REGION Network 16: AV Outlet
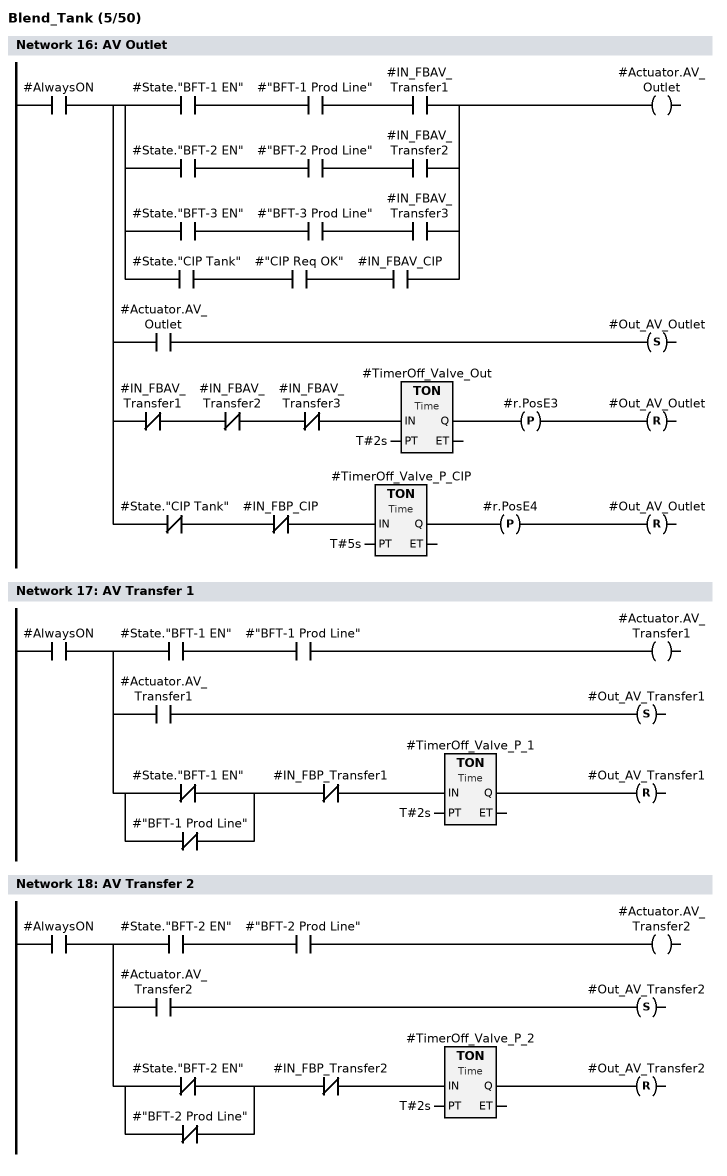
   RUNG wire#powerrail
      Contact( #AlwaysON )
      wire#w1
      Contact( #State."BFT-1 EN" )
      Contact( #"BFT-1 Prod Line" )
      Contact( #IN_FBAV_Transfer1 )
      wire#w2
      Coil( #Actuator.AV_Outlet )
   END_RUNG
   RUNG wire#w1
      Contact( #State."BFT-2 EN" )
      Contact( #"BFT-2 Prod Line" )
      Contact( #IN_FBAV_Transfer2 )
   END_RUNG wire#w2
   RUNG wire#w1
      Contact( #State."BFT-3 EN" )
      Contact( #"BFT-3 Prod Line" )
      Contact( #IN_FBAV_Transfer3 )
   END_RUNG wire#w2
   RUNG wire#w1
      Contact( #State."CIP Tank" )
      Contact( #"CIP Req OK" )
      Contact( #IN_FBAV_CIP )
   END_RUNG wire#w2
   RUNG wire#w1
      Contact( #Actuator.AV_Outlet )
      S_Coil( #Out_AV_Outlet )
   END_RUNG
   RUNG wire#w1
      I_Contact( #IN_FBAV_Transfer1 )
      I_Contact( #IN_FBAV_Transfer2 )
      I_Contact( #IN_FBAV_Transfer3 )
      { S7_Templates := "time_type := Time" } #TimerOff_Valve_Out.TON(pt := T#2s, et =>)
      P_Trig( #r.PosE3 )
      R_Coil( #Out_AV_Outlet )
   END_RUNG
   RUNG wire#w1
      I_Contact( #State."CIP Tank" )
      I_Contact( #IN_FBP_CIP )
      { S7_Templates := "time_type := Time" } #TimerOff_Valve_P_CIP.TON(pt := T#5s, et =>)
      P_Trig( #r.PosE4 )
      R_Coil( #Out_AV_Outlet )
   END_RUNG
   // the same network as SCL:
   #Actuator.AV_Outlet := #AlwaysON AND ((#State."BFT-1 EN" AND #"BFT-1 Prod Line" AND #IN_FBAV_Transfer1) OR (#State."BFT-2 EN" AND #"BFT-2 Prod Line" AND #IN_FBAV_Transfer2) OR (#State."BFT-3 EN" AND #"BFT-3 Prod Line" AND #IN_FBAV_Transfer3) OR (#State."CIP Tank" AND #"CIP Req OK" AND #IN_FBAV_CIP));
   IF #AlwaysON AND #Actuator.AV_Outlet THEN #Out_AV_Outlet := TRUE; END_IF;
   #TimerOff_Valve_Out(IN := #AlwaysON AND NOT #IN_FBAV_Transfer1 AND NOT #IN_FBAV_Transfer2 AND NOT #IN_FBAV_Transfer3,   // TON
                       PT := T#2s);
   #_w1 := #TimerOff_Valve_Out.Q AND NOT #r.PosE3;   // rising edge
   #r.PosE3 := #TimerOff_Valve_Out.Q;
   IF #_w1 THEN #Out_AV_Outlet := FALSE; END_IF;
   #TimerOff_Valve_P_CIP(IN := #AlwaysON AND NOT #State."CIP Tank" AND NOT #IN_FBP_CIP, PT := T#5s);   // TON
   #_w2 := #TimerOff_Valve_P_CIP.Q AND NOT #r.PosE4;   // rising edge
   #r.PosE4 := #TimerOff_Valve_P_CIP.Q;
   IF #_w2 THEN #Out_AV_Outlet := FALSE; END_IF;
END_REGION

REGION Network 17: AV Transfer 1
   RUNG wire#powerrail
      Contact( #AlwaysON )
      wire#w1
      Contact( #State."BFT-1 EN" )
      Contact( #"BFT-1 Prod Line" )
      Coil( #Actuator.AV_Transfer1 )
   END_RUNG
   RUNG wire#w1
      Contact( #Actuator.AV_Transfer1 )
      S_Coil( #Out_AV_Transfer1 )
   END_RUNG
   RUNG wire#w1
      I_Contact( #State."BFT-1 EN" )
      wire#w2
      I_Contact( #IN_FBP_Transfer1 )
      { S7_Templates := "time_type := Time" } #TimerOff_Valve_P_1.TON(pt := T#2s, et =>)
      R_Coil( #Out_AV_Transfer1 )
   END_RUNG
   RUNG wire#w1
      I_Contact( #"BFT-1 Prod Line" )
   END_RUNG wire#w2
   // the same network as SCL:
   #Actuator.AV_Transfer1 := #AlwaysON AND #State."BFT-1 EN" AND #"BFT-1 Prod Line";
   IF #AlwaysON AND #Actuator.AV_Transfer1 THEN #Out_AV_Transfer1 := TRUE; END_IF;
   #TimerOff_Valve_P_1(IN := #AlwaysON AND (NOT #State."BFT-1 EN" OR NOT #"BFT-1 Prod Line") AND NOT #IN_FBP_Transfer1,   // TON
                       PT := T#2s);
   IF #TimerOff_Valve_P_1.Q THEN #Out_AV_Transfer1 := FALSE; END_IF;
END_REGION

REGION Network 18: AV Transfer 2
   RUNG wire#powerrail
      Contact( #AlwaysON )
      wire#w1
      Contact( #State."BFT-2 EN" )
      Contact( #"BFT-2 Prod Line" )
      Coil( #Actuator.AV_Transfer2 )
   END_RUNG
   RUNG wire#w1
      Contact( #Actuator.AV_Transfer2 )
      S_Coil( #Out_AV_Transfer2 )
   END_RUNG
   RUNG wire#w1
      I_Contact( #State."BFT-2 EN" )
      wire#w2
      I_Contact( #IN_FBP_Transfer2 )
      { S7_Templates := "time_type := Time" } #TimerOff_Valve_P_2.TON(pt := T#2s, et =>)
      R_Coil( #Out_AV_Transfer2 )
   END_RUNG
   RUNG wire#w1
      I_Contact( #"BFT-2 Prod Line" )
   END_RUNG wire#w2
   // the same network as SCL:
   #Actuator.AV_Transfer2 := #AlwaysON AND #State."BFT-2 EN" AND #"BFT-2 Prod Line";
   IF #AlwaysON AND #Actuator.AV_Transfer2 THEN #Out_AV_Transfer2 := TRUE; END_IF;
   #TimerOff_Valve_P_2(IN := #AlwaysON AND (NOT #State."BFT-2 EN" OR NOT #"BFT-2 Prod Line") AND NOT #IN_FBP_Transfer2,   // TON
                       PT := T#2s);
   IF #TimerOff_Valve_P_2.Q THEN #Out_AV_Transfer2 := FALSE; END_IF;
END_REGION

REGION Network 19: AV Transfer 3
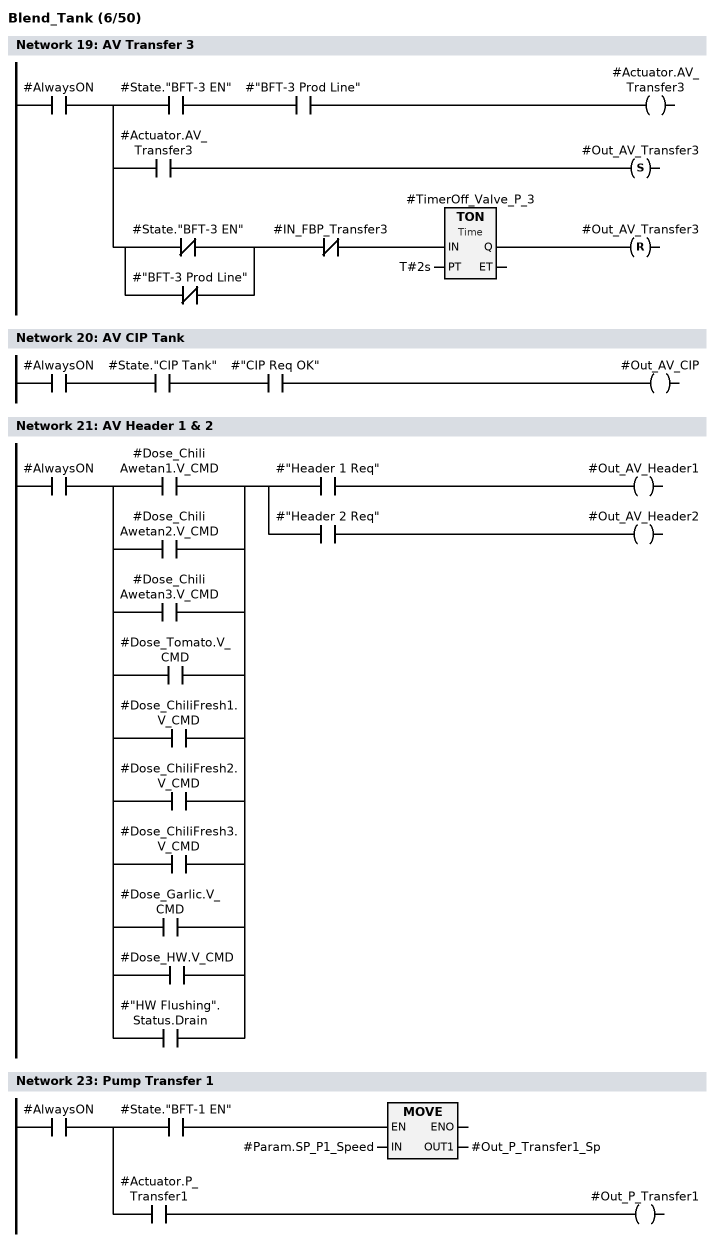
   RUNG wire#powerrail
      Contact( #AlwaysON )
      wire#w1
      Contact( #State."BFT-3 EN" )
      Contact( #"BFT-3 Prod Line" )
      Coil( #Actuator.AV_Transfer3 )
   END_RUNG
   RUNG wire#w1
      Contact( #Actuator.AV_Transfer3 )
      S_Coil( #Out_AV_Transfer3 )
   END_RUNG
   RUNG wire#w1
      I_Contact( #State."BFT-3 EN" )
      wire#w2
      I_Contact( #IN_FBP_Transfer3 )
      { S7_Templates := "time_type := Time" } #TimerOff_Valve_P_3.TON(pt := T#2s, et =>)
      R_Coil( #Out_AV_Transfer3 )
   END_RUNG
   RUNG wire#w1
      I_Contact( #"BFT-3 Prod Line" )
   END_RUNG wire#w2
   // the same network as SCL:
   #Actuator.AV_Transfer3 := #AlwaysON AND #State."BFT-3 EN" AND #"BFT-3 Prod Line";
   IF #AlwaysON AND #Actuator.AV_Transfer3 THEN #Out_AV_Transfer3 := TRUE; END_IF;
   #TimerOff_Valve_P_3(IN := #AlwaysON AND (NOT #State."BFT-3 EN" OR NOT #"BFT-3 Prod Line") AND NOT #IN_FBP_Transfer3,   // TON
                       PT := T#2s);
   IF #TimerOff_Valve_P_3.Q THEN #Out_AV_Transfer3 := FALSE; END_IF;
END_REGION

REGION Network 20: AV CIP Tank
   RUNG wire#powerrail
      Contact( #AlwaysON )
      Contact( #State."CIP Tank" )
      Contact( #"CIP Req OK" )
      Coil( #Out_AV_CIP )
   END_RUNG
   // the same network as SCL:
   #Out_AV_CIP := #AlwaysON AND #State."CIP Tank" AND #"CIP Req OK";
END_REGION

REGION Network 21: AV Header 1 & 2
   RUNG wire#powerrail
      Contact( #AlwaysON )
      wire#w1
      Contact( #Dose_ChiliAwetan1.V_CMD )
      wire#w2
      Contact( #"Header 1 Req" )
      Coil( #Out_AV_Header1 )
   END_RUNG
   RUNG wire#w1
      Contact( #Dose_ChiliAwetan2.V_CMD )
   END_RUNG wire#w2
   RUNG wire#w1
      Contact( #Dose_ChiliAwetan3.V_CMD )
   END_RUNG wire#w2
   RUNG wire#w1
      Contact( #Dose_Tomato.V_CMD )
   END_RUNG wire#w2
   RUNG wire#w1
      Contact( #Dose_ChiliFresh1.V_CMD )
   END_RUNG wire#w2
   RUNG wire#w1
      Contact( #Dose_ChiliFresh2.V_CMD )
   END_RUNG wire#w2
   RUNG wire#w1
      Contact( #Dose_ChiliFresh3.V_CMD )
   END_RUNG wire#w2
   RUNG wire#w1
      Contact( #Dose_Garlic.V_CMD )
   END_RUNG wire#w2
   RUNG wire#w1
      Contact( #Dose_HW.V_CMD )
   END_RUNG wire#w2
   RUNG wire#w1
      Contact( #"HW Flushing".Status.Drain )
   END_RUNG wire#w2
   RUNG wire#w2
      Contact( #"Header 2 Req" )
      Coil( #Out_AV_Header2 )
   END_RUNG
   // the same network as SCL:
   #_w1 := #AlwaysON AND (#Dose_ChiliAwetan1.V_CMD OR #Dose_ChiliAwetan2.V_CMD OR #Dose_ChiliAwetan3.V_CMD OR #Dose_Tomato.V_CMD OR #Dose_ChiliFresh1.V_CMD OR #Dose_ChiliFresh2.V_CMD OR #Dose_ChiliFresh3.V_CMD OR #Dose_Garlic.V_CMD OR #Dose_HW.V_CMD OR #"HW Flushing".Status.Drain);
   #Out_AV_Header1 := #_w1 AND #"Header 1 Req";
   #Out_AV_Header2 := #_w1 AND #"Header 2 Req";
END_REGION

REGION Network 23: Pump Transfer 1
   RUNG wire#powerrail
      Contact( #AlwaysON )
      wire#w1
      Contact( #State."BFT-1 EN" )
      Move(in := #Param.SP_P1_Speed, out1 => #Out_P_Transfer1_Sp)
   END_RUNG
   RUNG wire#w1
      Contact( #Actuator.P_Transfer1 )
      Coil( #Out_P_Transfer1 )
   END_RUNG
   // the same network as SCL:
   IF #AlwaysON AND #State."BFT-1 EN" THEN #Out_P_Transfer1_Sp := #Param.SP_P1_Speed; END_IF;
   #Out_P_Transfer1 := #AlwaysON AND #Actuator.P_Transfer1;
END_REGION

REGION Network 24: Pump Transfer 2
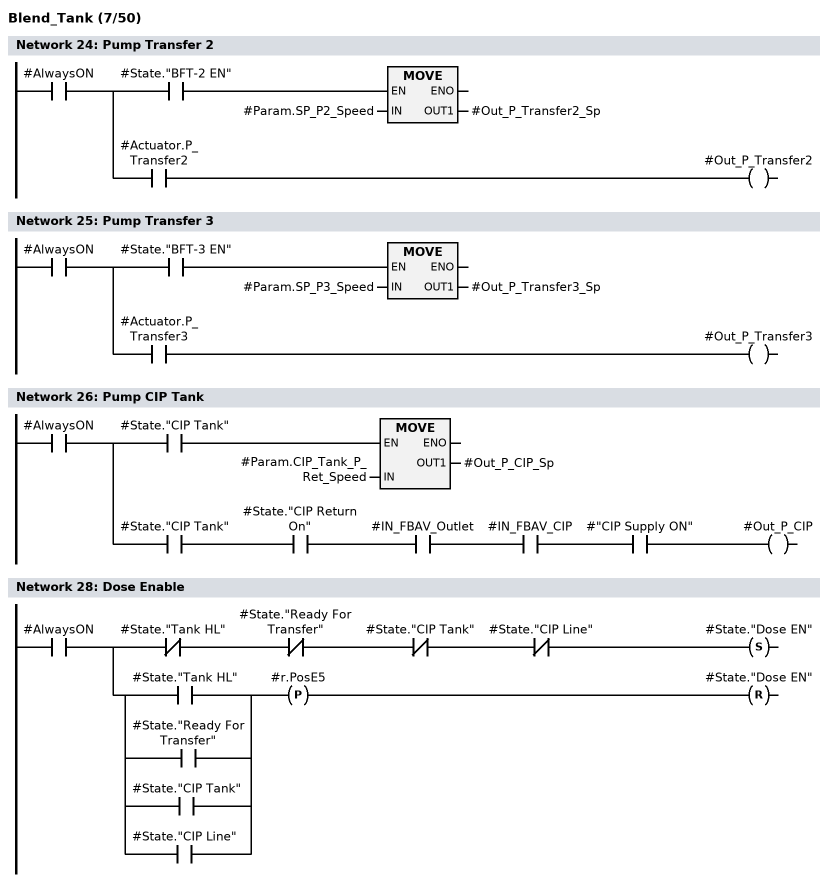
   RUNG wire#powerrail
      Contact( #AlwaysON )
      wire#w1
      Contact( #State."BFT-2 EN" )
      Move(in := #Param.SP_P2_Speed, out1 => #Out_P_Transfer2_Sp)
   END_RUNG
   RUNG wire#w1
      Contact( #Actuator.P_Transfer2 )
      Coil( #Out_P_Transfer2 )
   END_RUNG
   // the same network as SCL:
   IF #AlwaysON AND #State."BFT-2 EN" THEN #Out_P_Transfer2_Sp := #Param.SP_P2_Speed; END_IF;
   #Out_P_Transfer2 := #AlwaysON AND #Actuator.P_Transfer2;
END_REGION

REGION Network 25: Pump Transfer 3
   RUNG wire#powerrail
      Contact( #AlwaysON )
      wire#w1
      Contact( #State."BFT-3 EN" )
      Move(in := #Param.SP_P3_Speed, out1 => #Out_P_Transfer3_Sp)
   END_RUNG
   RUNG wire#w1
      Contact( #Actuator.P_Transfer3 )
      Coil( #Out_P_Transfer3 )
   END_RUNG
   // the same network as SCL:
   IF #AlwaysON AND #State."BFT-3 EN" THEN #Out_P_Transfer3_Sp := #Param.SP_P3_Speed; END_IF;
   #Out_P_Transfer3 := #AlwaysON AND #Actuator.P_Transfer3;
END_REGION

REGION Network 26: Pump CIP Tank
   RUNG wire#powerrail
      Contact( #AlwaysON )
      wire#w1
      Contact( #State."CIP Tank" )
      Move(in := #Param.CIP_Tank_P_Ret_Speed, out1 => #Out_P_CIP_Sp)
   END_RUNG
   RUNG wire#w1
      Contact( #State."CIP Tank" )
      Contact( #State."CIP Return On" )
      Contact( #IN_FBAV_Outlet )
      Contact( #IN_FBAV_CIP )
      Contact( #"CIP Supply ON" )
      Coil( #Out_P_CIP )
   END_RUNG
   // the same network as SCL:
   IF #AlwaysON AND #State."CIP Tank" THEN #Out_P_CIP_Sp := #Param.CIP_Tank_P_Ret_Speed; END_IF;
   #Out_P_CIP := #AlwaysON AND #State."CIP Tank" AND #State."CIP Return On" AND #IN_FBAV_Outlet AND #IN_FBAV_CIP AND #"CIP Supply ON";
END_REGION

REGION Network 28: Dose Enable
   RUNG wire#powerrail
      Contact( #AlwaysON )
      wire#w1
      I_Contact( #State."Tank HL" )
      I_Contact( #State."Ready For Transfer" )
      I_Contact( #State."CIP Tank" )
      I_Contact( #State."CIP Line" )
      S_Coil( #State."Dose EN" )
   END_RUNG
   RUNG wire#w1
      Contact( #State."Tank HL" )
      wire#w2
      P_Trig( #r.PosE5 )
      R_Coil( #State."Dose EN" )
   END_RUNG
   RUNG wire#w1
      Contact( #State."Ready For Transfer" )
   END_RUNG wire#w2
   RUNG wire#w1
      Contact( #State."CIP Tank" )
   END_RUNG wire#w2
   RUNG wire#w1
      Contact( #State."CIP Line" )
   END_RUNG wire#w2
   // the same network as SCL:
   IF #AlwaysON AND NOT #State."Tank HL" AND NOT #State."Ready For Transfer" AND NOT #State."CIP Tank" AND NOT #State."CIP Line" THEN
       #State."Dose EN" := TRUE;
   END_IF;
   #_w1 := #AlwaysON AND (#State."Tank HL" OR #State."Ready For Transfer" OR #State."CIP Tank" OR #State."CIP Line");
   #_w2 := #_w1 AND NOT #r.PosE5;   // rising edge
   #r.PosE5 := #_w1;
   IF #_w2 THEN #State."Dose EN" := FALSE; END_IF;
END_REGION

NETWORK
TITLE = Raw Material & Tank Dose State
// Raw Material Dose State
      O     #Dose_ChiliAwetan1.QDOSERun;
      O     #Dose_ChiliAwetan2.QDOSERun;
      O     #Dose_ChiliAwetan3.QDOSERun;
      O     #Dose_Tomato.QDOSERun;
      O     #Dose_ChiliFresh1.QDOSERun;
      O     #Dose_ChiliFresh2.QDOSERun;
      O     #Dose_ChiliFresh3.QDOSERun;
      O     #Dose_Garlic.QDOSERun;
      O     #Dose_HW.QDOSERun;
      =     #State."RM Dose";

// Dose Run State
      O     #State."RM Dose";
      O     #Dose_Vinegar.QDOSERun;
      O     #Dose_Sugar.QDOSERun;
      O     #Dose_Salt.QDOSERun;
      O     #Dose_ProWater.QDOSERun;
      O     #Dose_Homomixer.QDOSERun;
      =     #State."Dose On Prog";


REGION Network 31: Header 1 & 2 --- Vinegar --- Sugar --- Salt --- ProWater --- Homomixer Enable
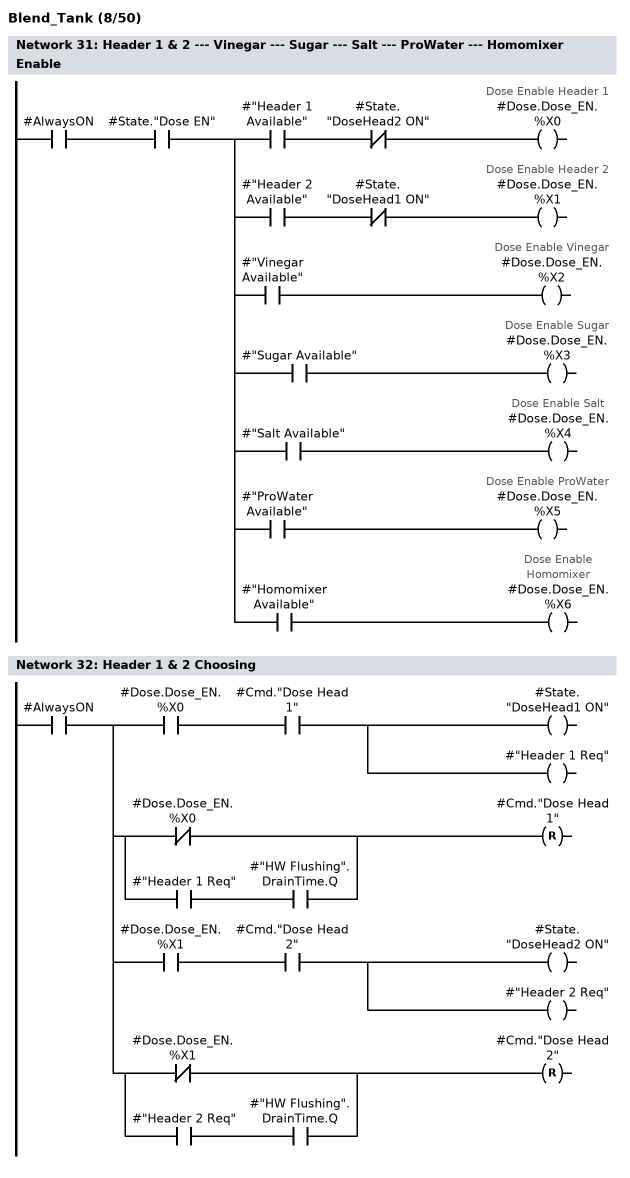
   RUNG wire#powerrail
      Contact( #AlwaysON )
      Contact( #State."Dose EN" )
      wire#w1
      Contact( #"Header 1 Available" )
      I_Contact( #State."DoseHead2 ON" )
      Coil( #Dose.Dose_EN.%X0 )   // Dose Enable Header 1
   END_RUNG
   RUNG wire#w1
      Contact( #"Header 2 Available" )
      I_Contact( #State."DoseHead1 ON" )
      Coil( #Dose.Dose_EN.%X1 )   // Dose Enable Header 2
   END_RUNG
   RUNG wire#w1
      Contact( #"Vinegar Available" )
      Coil( #Dose.Dose_EN.%X2 )   // Dose Enable Vinegar
   END_RUNG
   RUNG wire#w1
      Contact( #"Sugar Available" )
      Coil( #Dose.Dose_EN.%X3 )   // Dose Enable Sugar
   END_RUNG
   RUNG wire#w1
      Contact( #"Salt Available" )
      Coil( #Dose.Dose_EN.%X4 )   // Dose Enable Salt
   END_RUNG
   RUNG wire#w1
      Contact( #"ProWater Available" )
      Coil( #Dose.Dose_EN.%X5 )   // Dose Enable ProWater
   END_RUNG
   RUNG wire#w1
      Contact( #"Homomixer Available" )
      Coil( #Dose.Dose_EN.%X6 )   // Dose Enable Homomixer
   END_RUNG
   // the same network as SCL:
   #_w1 := #AlwaysON AND #State."Dose EN";
   #Dose.Dose_EN.%X0 := #_w1 AND #"Header 1 Available" AND NOT #State."DoseHead2 ON";   // Dose Enable Header 1
   #Dose.Dose_EN.%X1 := #_w1 AND #"Header 2 Available" AND NOT #State."DoseHead1 ON";   // Dose Enable Header 2
   #Dose.Dose_EN.%X2 := #_w1 AND #"Vinegar Available";   // Dose Enable Vinegar
   #Dose.Dose_EN.%X3 := #_w1 AND #"Sugar Available";   // Dose Enable Sugar
   #Dose.Dose_EN.%X4 := #_w1 AND #"Salt Available";   // Dose Enable Salt
   #Dose.Dose_EN.%X5 := #_w1 AND #"ProWater Available";   // Dose Enable ProWater
   #Dose.Dose_EN.%X6 := #_w1 AND #"Homomixer Available";   // Dose Enable Homomixer
END_REGION

REGION Network 32: Header 1 & 2 Choosing
   RUNG wire#powerrail
      Contact( #AlwaysON )
      wire#w1
      Contact( #Dose.Dose_EN.%X0 )
      Contact( #Cmd."Dose Head 1" )
      wire#w2
      Coil( #State."DoseHead1 ON" )
   END_RUNG
   RUNG wire#w2
      Coil( #"Header 1 Req" )
   END_RUNG
   RUNG wire#w1
      I_Contact( #Dose.Dose_EN.%X0 )
      wire#w3
      R_Coil( #Cmd."Dose Head 1" )
   END_RUNG
   RUNG wire#w1
      Contact( #"Header 1 Req" )
      Contact( #"HW Flushing".DrainTime.Q )
   END_RUNG wire#w3
   RUNG wire#w1
      Contact( #Dose.Dose_EN.%X1 )
      Contact( #Cmd."Dose Head 2" )
      wire#w4
      Coil( #State."DoseHead2 ON" )
   END_RUNG
   RUNG wire#w4
      Coil( #"Header 2 Req" )
   END_RUNG
   RUNG wire#w1
      I_Contact( #Dose.Dose_EN.%X1 )
      wire#w5
      R_Coil( #Cmd."Dose Head 2" )
   END_RUNG
   RUNG wire#w1
      Contact( #"Header 2 Req" )
      Contact( #"HW Flushing".DrainTime.Q )
   END_RUNG wire#w5
   // the same network as SCL:
   #State."DoseHead1 ON" := #AlwaysON AND #Dose.Dose_EN.%X0 AND #Cmd."Dose Head 1";
   #"Header 1 Req" := #State."DoseHead1 ON";
   IF #AlwaysON AND (NOT #Dose.Dose_EN.%X0 OR (#"Header 1 Req" AND #"HW Flushing".DrainTime.Q)) THEN
       #Cmd."Dose Head 1" := FALSE;
   END_IF;
   #State."DoseHead2 ON" := #AlwaysON AND #Dose.Dose_EN.%X1 AND #Cmd."Dose Head 2";
   #"Header 2 Req" := #State."DoseHead2 ON";
   IF #AlwaysON AND (NOT #Dose.Dose_EN.%X1 OR (#"Header 2 Req" AND #"HW Flushing".DrainTime.Q)) THEN
       #Cmd."Dose Head 2" := FALSE;
   END_IF;
END_REGION

NETWORK
TITLE = Header 1 & 2 Request
// Header 1 Request
//      O     #Dose.Dose_Header_Req.%X0// ChiliAwetan1 Header1 Req
//      O     #Dose.Dose_Header_Req.%X1// ChiliAwetan2 Header1 Req
//      O     #Dose.Dose_Header_Req.%X2// ChiliAwetan3 Header1 Req
//      O     #Dose.Dose_Header_Req.%X3// Tomato Header1 Req
//      O     #Dose.Dose_Header_Req.%X4// ChiliFresh1 Header1 Req
//      O     #Dose.Dose_Header_Req.%X5// ChiliFresh2 Header1 Req
//      O     #Dose.Dose_Header_Req.%X6// ChiliFresh3 Header1 Req
//      O     #Dose.Dose_Header_Req.%X7// Garlic Header1 Req
//      O     #Dose.Dose_Header_Req.%X8// HotWater Header1 Req
//     =     #"Header 1 Req"

// Header 2 Request
//      O     #Dose.Dose_Header_Req.%X16// ChiliAwetan1 Header2 Req
//      O     #Dose.Dose_Header_Req.%X17// ChiliAwetan2 Header2 Req
//      O     #Dose.Dose_Header_Req.%X18// ChiliAwetan3 Header2 Req
//      O     #Dose.Dose_Header_Req.%X19// Tomato Header2 Req
//      O     #Dose.Dose_Header_Req.%X20// ChiliFresh1 Header2 Req
//      O     #Dose.Dose_Header_Req.%X21// ChiliFresh2 Header2 Req
//      O     #Dose.Dose_Header_Req.%X22// ChiliFresh3 Header2 Req
//      O     #Dose.Dose_Header_Req.%X23// Garlic Header2 Req
//      O     #Dose.Dose_Header_Req.%X24// HotWater Header2 Req
//      =     #"Header 2 Req"


REGION Network 36: ChiliAwetan1 Setpoint
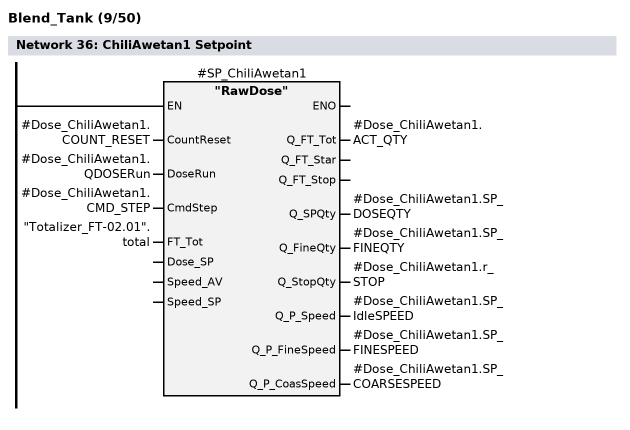
   RUNG wire#powerrail
      #SP_ChiliAwetan1(CountReset := #Dose_ChiliAwetan1.COUNT_RESET, DoseRun := #Dose_ChiliAwetan1.QDOSERun, CmdStep := #Dose_ChiliAwetan1.CMD_STEP, FT_Tot := "Totalizer_FT-02.01".total, Dose_SP :=, Speed_AV :=, Speed_SP :=, Q_FT_Tot => #Dose_ChiliAwetan1.ACT_QTY, Q_FT_Star =>, Q_FT_Stop =>, Q_SPQty => #Dose_ChiliAwetan1.SP_DOSEQTY, Q_FineQty => #Dose_ChiliAwetan1.SP_FINEQTY, Q_StopQty => #Dose_ChiliAwetan1.r_STOP, Q_P_Speed => #Dose_ChiliAwetan1.SP_IdleSPEED, Q_P_FineSpeed => #Dose_ChiliAwetan1.SP_FINESPEED, Q_P_CoasSpeed => #Dose_ChiliAwetan1.SP_COARSESPEED)
   END_RUNG
   // the same network as SCL:
   #SP_ChiliAwetan1(CountReset := #Dose_ChiliAwetan1.COUNT_RESET,   // "RawDose"
                    DoseRun := #Dose_ChiliAwetan1.QDOSERun,
                    CmdStep := #Dose_ChiliAwetan1.CMD_STEP,
                    FT_Tot := "Totalizer_FT-02.01".total,
                    Q_FT_Tot => #Dose_ChiliAwetan1.ACT_QTY,
                    Q_SPQty => #Dose_ChiliAwetan1.SP_DOSEQTY,
                    Q_FineQty => #Dose_ChiliAwetan1.SP_FINEQTY,
                    Q_StopQty => #Dose_ChiliAwetan1.r_STOP,
                    Q_P_Speed => #Dose_ChiliAwetan1.SP_IdleSPEED,
                    Q_P_FineSpeed => #Dose_ChiliAwetan1.SP_FINESPEED,
                    Q_P_CoasSpeed => #Dose_ChiliAwetan1.SP_COARSESPEED);
END_REGION

REGION Network 37: Command Dose ChiliAwetan1
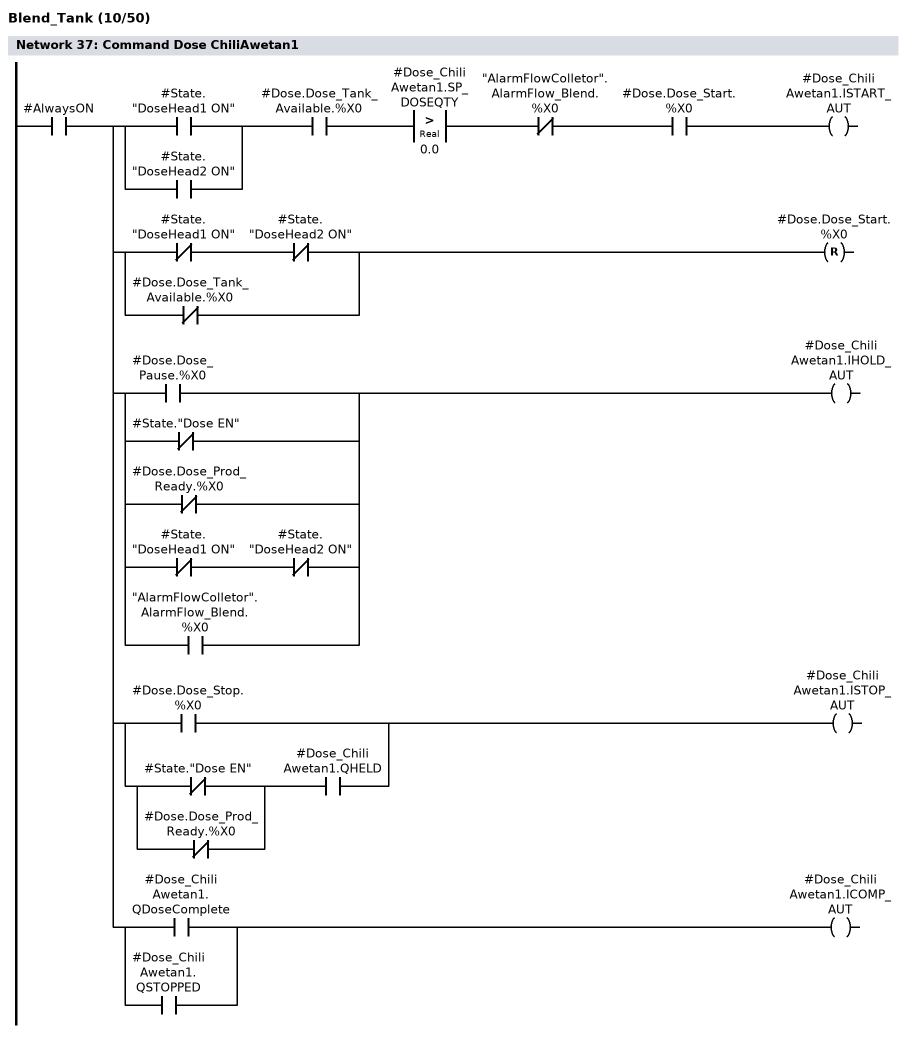
   RUNG wire#powerrail
      Contact( #AlwaysON )
      wire#w1
      Contact( #State."DoseHead1 ON" )
      wire#w2
      Contact( #Dose.Dose_Tank_Available.%X0 )
      { S7_Templates := "SrcType := Real" } GT_Contact(in1 := #Dose_ChiliAwetan1.SP_DOSEQTY, in2 := 0.0)
      I_Contact( "AlarmFlowColletor".AlarmFlow_Blend.%X0 )
      Contact( #Dose.Dose_Start.%X0 )
      Coil( #Dose_ChiliAwetan1.ISTART_AUT )
   END_RUNG
   RUNG wire#w1
      Contact( #State."DoseHead2 ON" )
   END_RUNG wire#w2
   RUNG wire#w1
      I_Contact( #State."DoseHead1 ON" )
      I_Contact( #State."DoseHead2 ON" )
      wire#w3
      R_Coil( #Dose.Dose_Start.%X0 )
   END_RUNG
   RUNG wire#w1
      I_Contact( #Dose.Dose_Tank_Available.%X0 )
   END_RUNG wire#w3
   RUNG wire#w1
      Contact( #Dose.Dose_Pause.%X0 )
      wire#w4
      Coil( #Dose_ChiliAwetan1.IHOLD_AUT )
   END_RUNG
   RUNG wire#w1
      I_Contact( #State."Dose EN" )
   END_RUNG wire#w4
   RUNG wire#w1
      I_Contact( #Dose.Dose_Prod_Ready.%X0 )
   END_RUNG wire#w4
   RUNG wire#w1
      I_Contact( #State."DoseHead1 ON" )
      I_Contact( #State."DoseHead2 ON" )
   END_RUNG wire#w4
   RUNG wire#w1
      Contact( "AlarmFlowColletor".AlarmFlow_Blend.%X0 )
   END_RUNG wire#w4
   RUNG wire#w1
      Contact( #Dose.Dose_Stop.%X0 )
      wire#w5
      Coil( #Dose_ChiliAwetan1.ISTOP_AUT )
   END_RUNG
   RUNG wire#w1
      I_Contact( #State."Dose EN" )
      wire#w6
      Contact( #Dose_ChiliAwetan1.QHELD )
   END_RUNG wire#w5
   RUNG wire#w1
      I_Contact( #Dose.Dose_Prod_Ready.%X0 )
   END_RUNG wire#w6
   RUNG wire#w1
      Contact( #Dose_ChiliAwetan1.QDoseComplete )
      wire#w7
      Coil( #Dose_ChiliAwetan1.ICOMP_AUT )
   END_RUNG
   RUNG wire#w1
      Contact( #Dose_ChiliAwetan1.QSTOPPED )
   END_RUNG wire#w7
   // the same network as SCL:
   #Dose_ChiliAwetan1.ISTART_AUT := #AlwaysON AND (#State."DoseHead1 ON" OR #State."DoseHead2 ON") AND #Dose.Dose_Tank_Available.%X0 AND (#Dose_ChiliAwetan1.SP_DOSEQTY > 0.0) AND NOT "AlarmFlowColletor".AlarmFlow_Blend.%X0 AND #Dose.Dose_Start.%X0;
   IF #AlwaysON AND ((NOT #State."DoseHead1 ON" AND NOT #State."DoseHead2 ON") OR NOT #Dose.Dose_Tank_Available.%X0) THEN
       #Dose.Dose_Start.%X0 := FALSE;
   END_IF;
   #Dose_ChiliAwetan1.IHOLD_AUT := #AlwaysON AND (#Dose.Dose_Pause.%X0 OR NOT #State."Dose EN" OR NOT #Dose.Dose_Prod_Ready.%X0 OR (NOT #State."DoseHead1 ON" AND NOT #State."DoseHead2 ON") OR "AlarmFlowColletor".AlarmFlow_Blend.%X0);
   #Dose_ChiliAwetan1.ISTOP_AUT := #AlwaysON AND (#Dose.Dose_Stop.%X0 OR ((NOT #State."Dose EN" OR NOT #Dose.Dose_Prod_Ready.%X0) AND #Dose_ChiliAwetan1.QHELD));
   #Dose_ChiliAwetan1.ICOMP_AUT := #AlwaysON AND (#Dose_ChiliAwetan1.QDoseComplete OR #Dose_ChiliAwetan1.QSTOPPED);
END_REGION

REGION Network 38: Dose ChiliAwetan1
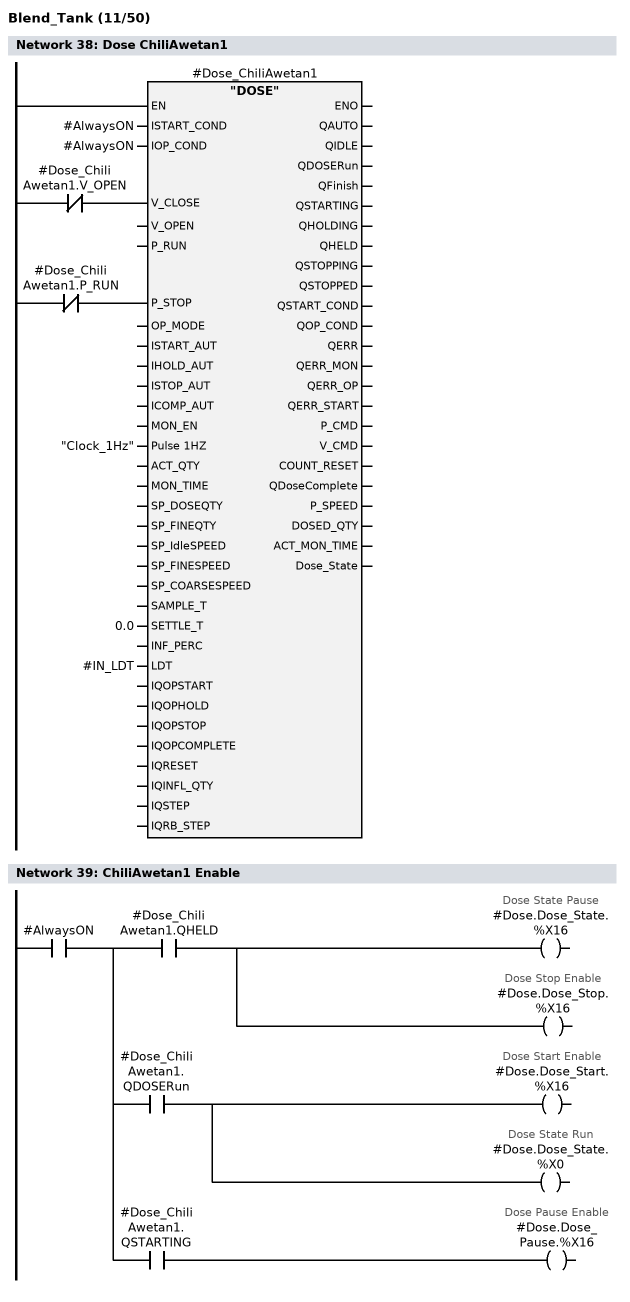
   RUNG wire#powerrail
      #Dose_ChiliAwetan1(V_CLOSE := wire#w1, P_STOP := wire#w2, ISTART_COND := #AlwaysON, IOP_COND := #AlwaysON, V_OPEN :=, P_RUN :=, OP_MODE :=, ISTART_AUT :=, IHOLD_AUT :=, ISTOP_AUT :=, ICOMP_AUT :=, MON_EN :=, "Pulse 1HZ" := "Clock_1Hz", ACT_QTY :=, MON_TIME :=, SP_DOSEQTY :=, SP_FINEQTY :=, SP_IdleSPEED :=, SP_FINESPEED :=, SP_COARSESPEED :=, SAMPLE_T :=, SETTLE_T := 0.0, INF_PERC :=, LDT := #IN_LDT, IQOPSTART :=, IQOPHOLD :=, IQOPSTOP :=, IQOPCOMPLETE :=, IQRESET :=, IQINFL_QTY :=, IQSTEP :=, IQRB_STEP :=, QAUTO =>, QIDLE =>, QDOSERun =>, QFinish =>, QSTARTING =>, QHOLDING =>, QHELD =>, QSTOPPING =>, QSTOPPED =>, QSTART_COND =>, QOP_COND =>, QERR =>, QERR_MON =>, QERR_OP =>, QERR_START =>, P_CMD =>, V_CMD =>, COUNT_RESET =>, QDoseComplete =>, P_SPEED =>, DOSED_QTY =>, ACT_MON_TIME =>, Dose_State =>)
   END_RUNG
   RUNG wire#powerrail
      I_Contact( #Dose_ChiliAwetan1.V_OPEN )
   END_RUNG wire#w1
   RUNG wire#powerrail
      I_Contact( #Dose_ChiliAwetan1.P_RUN )
   END_RUNG wire#w2
   // the same network as SCL:
   #Dose_ChiliAwetan1(ISTART_COND := #AlwaysON,   // "DOSE"
                      IOP_COND := #AlwaysON,
                      V_CLOSE := NOT #Dose_ChiliAwetan1.V_OPEN,
                      P_STOP := NOT #Dose_ChiliAwetan1.P_RUN,
                      "Pulse 1HZ" := "Clock_1Hz",
                      SETTLE_T := 0.0,
                      LDT := #IN_LDT);
END_REGION

REGION Network 39: ChiliAwetan1 Enable
   RUNG wire#powerrail
      Contact( #AlwaysON )
      wire#w1
      Contact( #Dose_ChiliAwetan1.QHELD )
      wire#w2
      Coil( #Dose.Dose_State.%X16 )   // Dose State Pause
   END_RUNG
   RUNG wire#w2
      Coil( #Dose.Dose_Stop.%X16 )   // Dose Stop Enable
   END_RUNG
   RUNG wire#w1
      Contact( #Dose_ChiliAwetan1.QDOSERun )
      wire#w3
      Coil( #Dose.Dose_Start.%X16 )   // Dose Start Enable
   END_RUNG
   RUNG wire#w3
      Coil( #Dose.Dose_State.%X0 )   // Dose State Run
   END_RUNG
   RUNG wire#w1
      Contact( #Dose_ChiliAwetan1.QSTARTING )
      Coil( #Dose.Dose_Pause.%X16 )   // Dose Pause Enable
   END_RUNG
   // the same network as SCL:
   #Dose.Dose_State.%X16 := #AlwaysON AND #Dose_ChiliAwetan1.QHELD;   // Dose State Pause
   #Dose.Dose_Stop.%X16 := #Dose.Dose_State.%X16;   // Dose Stop Enable
   #Dose.Dose_Start.%X16 := #AlwaysON AND #Dose_ChiliAwetan1.QDOSERun;   // Dose Start Enable
   #Dose.Dose_State.%X0 := #Dose.Dose_Start.%X16;   // Dose State Run
   #Dose.Dose_Pause.%X16 := #AlwaysON AND #Dose_ChiliAwetan1.QSTARTING;   // Dose Pause Enable
END_REGION

REGION Network 40: ChiliAwetan1 Header Req
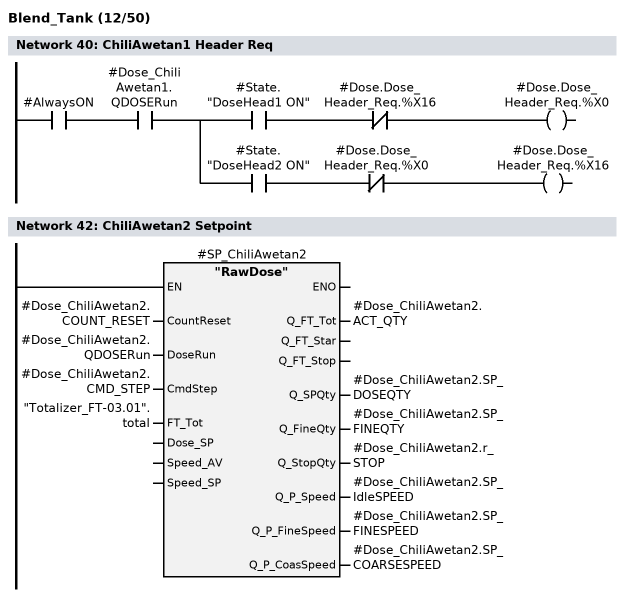
   RUNG wire#powerrail
      Contact( #AlwaysON )
      Contact( #Dose_ChiliAwetan1.QDOSERun )
      wire#w1
      Contact( #State."DoseHead1 ON" )
      I_Contact( #Dose.Dose_Header_Req.%X16 )
      Coil( #Dose.Dose_Header_Req.%X0 )
   END_RUNG
   RUNG wire#w1
      Contact( #State."DoseHead2 ON" )
      I_Contact( #Dose.Dose_Header_Req.%X0 )
      Coil( #Dose.Dose_Header_Req.%X16 )
   END_RUNG
   // the same network as SCL:
   #_w1 := #AlwaysON AND #Dose_ChiliAwetan1.QDOSERun;
   #Dose.Dose_Header_Req.%X0 := #_w1 AND #State."DoseHead1 ON" AND NOT #Dose.Dose_Header_Req.%X16;
   #Dose.Dose_Header_Req.%X16 := #_w1 AND #State."DoseHead2 ON" AND NOT #Dose.Dose_Header_Req.%X0;
END_REGION

REGION Network 42: ChiliAwetan2 Setpoint
   RUNG wire#powerrail
      #SP_ChiliAwetan2(CountReset := #Dose_ChiliAwetan2.COUNT_RESET, DoseRun := #Dose_ChiliAwetan2.QDOSERun, CmdStep := #Dose_ChiliAwetan2.CMD_STEP, FT_Tot := "Totalizer_FT-03.01".total, Dose_SP :=, Speed_AV :=, Speed_SP :=, Q_FT_Tot => #Dose_ChiliAwetan2.ACT_QTY, Q_FT_Star =>, Q_FT_Stop =>, Q_SPQty => #Dose_ChiliAwetan2.SP_DOSEQTY, Q_FineQty => #Dose_ChiliAwetan2.SP_FINEQTY, Q_StopQty => #Dose_ChiliAwetan2.r_STOP, Q_P_Speed => #Dose_ChiliAwetan2.SP_IdleSPEED, Q_P_FineSpeed => #Dose_ChiliAwetan2.SP_FINESPEED, Q_P_CoasSpeed => #Dose_ChiliAwetan2.SP_COARSESPEED)
   END_RUNG
   // the same network as SCL:
   #SP_ChiliAwetan2(CountReset := #Dose_ChiliAwetan2.COUNT_RESET,   // "RawDose"
                    DoseRun := #Dose_ChiliAwetan2.QDOSERun,
                    CmdStep := #Dose_ChiliAwetan2.CMD_STEP,
                    FT_Tot := "Totalizer_FT-03.01".total,
                    Q_FT_Tot => #Dose_ChiliAwetan2.ACT_QTY,
                    Q_SPQty => #Dose_ChiliAwetan2.SP_DOSEQTY,
                    Q_FineQty => #Dose_ChiliAwetan2.SP_FINEQTY,
                    Q_StopQty => #Dose_ChiliAwetan2.r_STOP,
                    Q_P_Speed => #Dose_ChiliAwetan2.SP_IdleSPEED,
                    Q_P_FineSpeed => #Dose_ChiliAwetan2.SP_FINESPEED,
                    Q_P_CoasSpeed => #Dose_ChiliAwetan2.SP_COARSESPEED);
END_REGION

REGION Network 43: Command Dose ChiliAwetan2
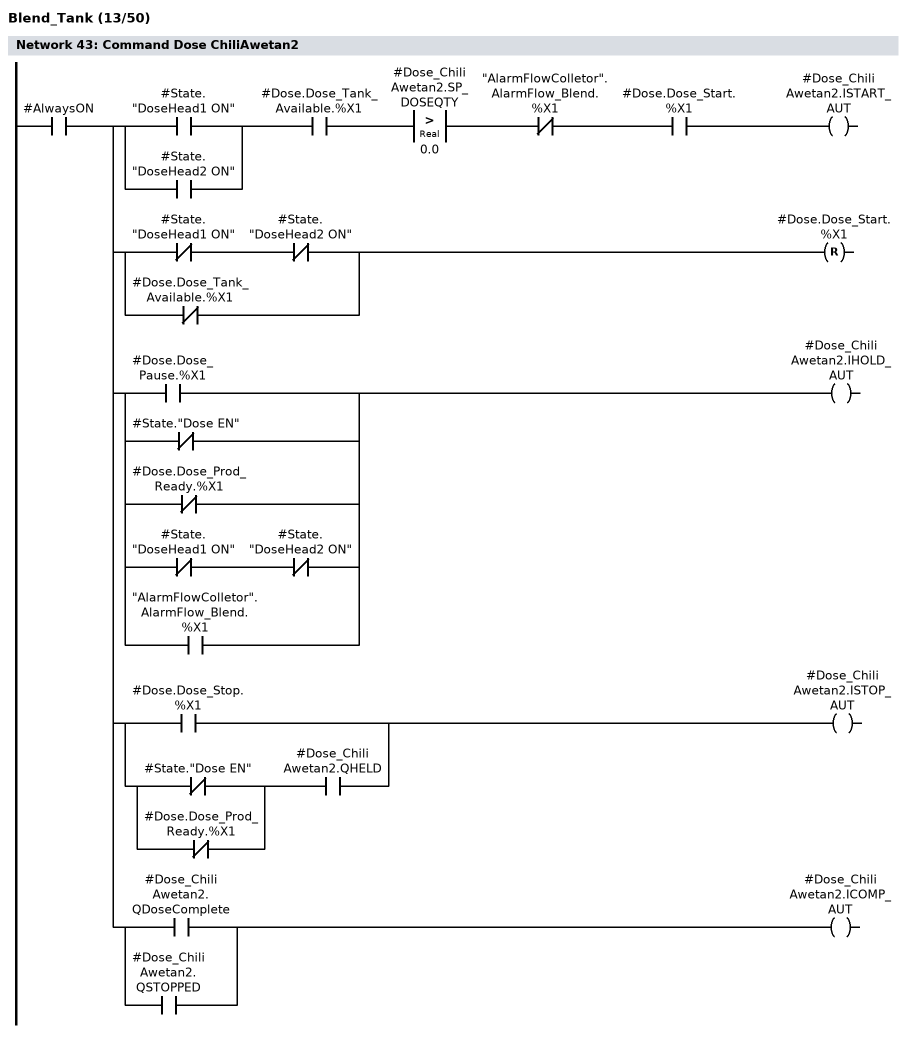
   RUNG wire#powerrail
      Contact( #AlwaysON )
      wire#w1
      Contact( #State."DoseHead1 ON" )
      wire#w2
      Contact( #Dose.Dose_Tank_Available.%X1 )
      { S7_Templates := "SrcType := Real" } GT_Contact(in1 := #Dose_ChiliAwetan2.SP_DOSEQTY, in2 := 0.0)
      I_Contact( "AlarmFlowColletor".AlarmFlow_Blend.%X1 )
      Contact( #Dose.Dose_Start.%X1 )
      Coil( #Dose_ChiliAwetan2.ISTART_AUT )
   END_RUNG
   RUNG wire#w1
      Contact( #State."DoseHead2 ON" )
   END_RUNG wire#w2
   RUNG wire#w1
      I_Contact( #State."DoseHead1 ON" )
      I_Contact( #State."DoseHead2 ON" )
      wire#w3
      R_Coil( #Dose.Dose_Start.%X1 )
   END_RUNG
   RUNG wire#w1
      I_Contact( #Dose.Dose_Tank_Available.%X1 )
   END_RUNG wire#w3
   RUNG wire#w1
      Contact( #Dose.Dose_Pause.%X1 )
      wire#w4
      Coil( #Dose_ChiliAwetan2.IHOLD_AUT )
   END_RUNG
   RUNG wire#w1
      I_Contact( #State."Dose EN" )
   END_RUNG wire#w4
   RUNG wire#w1
      I_Contact( #Dose.Dose_Prod_Ready.%X1 )
   END_RUNG wire#w4
   RUNG wire#w1
      I_Contact( #State."DoseHead1 ON" )
      I_Contact( #State."DoseHead2 ON" )
   END_RUNG wire#w4
   RUNG wire#w1
      Contact( "AlarmFlowColletor".AlarmFlow_Blend.%X1 )
   END_RUNG wire#w4
   RUNG wire#w1
      Contact( #Dose.Dose_Stop.%X1 )
      wire#w5
      Coil( #Dose_ChiliAwetan2.ISTOP_AUT )
   END_RUNG
   RUNG wire#w1
      I_Contact( #State."Dose EN" )
      wire#w6
      Contact( #Dose_ChiliAwetan2.QHELD )
   END_RUNG wire#w5
   RUNG wire#w1
      I_Contact( #Dose.Dose_Prod_Ready.%X1 )
   END_RUNG wire#w6
   RUNG wire#w1
      Contact( #Dose_ChiliAwetan2.QDoseComplete )
      wire#w7
      Coil( #Dose_ChiliAwetan2.ICOMP_AUT )
   END_RUNG
   RUNG wire#w1
      Contact( #Dose_ChiliAwetan2.QSTOPPED )
   END_RUNG wire#w7
   // the same network as SCL:
   #Dose_ChiliAwetan2.ISTART_AUT := #AlwaysON AND (#State."DoseHead1 ON" OR #State."DoseHead2 ON") AND #Dose.Dose_Tank_Available.%X1 AND (#Dose_ChiliAwetan2.SP_DOSEQTY > 0.0) AND NOT "AlarmFlowColletor".AlarmFlow_Blend.%X1 AND #Dose.Dose_Start.%X1;
   IF #AlwaysON AND ((NOT #State."DoseHead1 ON" AND NOT #State."DoseHead2 ON") OR NOT #Dose.Dose_Tank_Available.%X1) THEN
       #Dose.Dose_Start.%X1 := FALSE;
   END_IF;
   #Dose_ChiliAwetan2.IHOLD_AUT := #AlwaysON AND (#Dose.Dose_Pause.%X1 OR NOT #State."Dose EN" OR NOT #Dose.Dose_Prod_Ready.%X1 OR (NOT #State."DoseHead1 ON" AND NOT #State."DoseHead2 ON") OR "AlarmFlowColletor".AlarmFlow_Blend.%X1);
   #Dose_ChiliAwetan2.ISTOP_AUT := #AlwaysON AND (#Dose.Dose_Stop.%X1 OR ((NOT #State."Dose EN" OR NOT #Dose.Dose_Prod_Ready.%X1) AND #Dose_ChiliAwetan2.QHELD));
   #Dose_ChiliAwetan2.ICOMP_AUT := #AlwaysON AND (#Dose_ChiliAwetan2.QDoseComplete OR #Dose_ChiliAwetan2.QSTOPPED);
END_REGION

REGION Network 44: Dose ChiliAwetan2
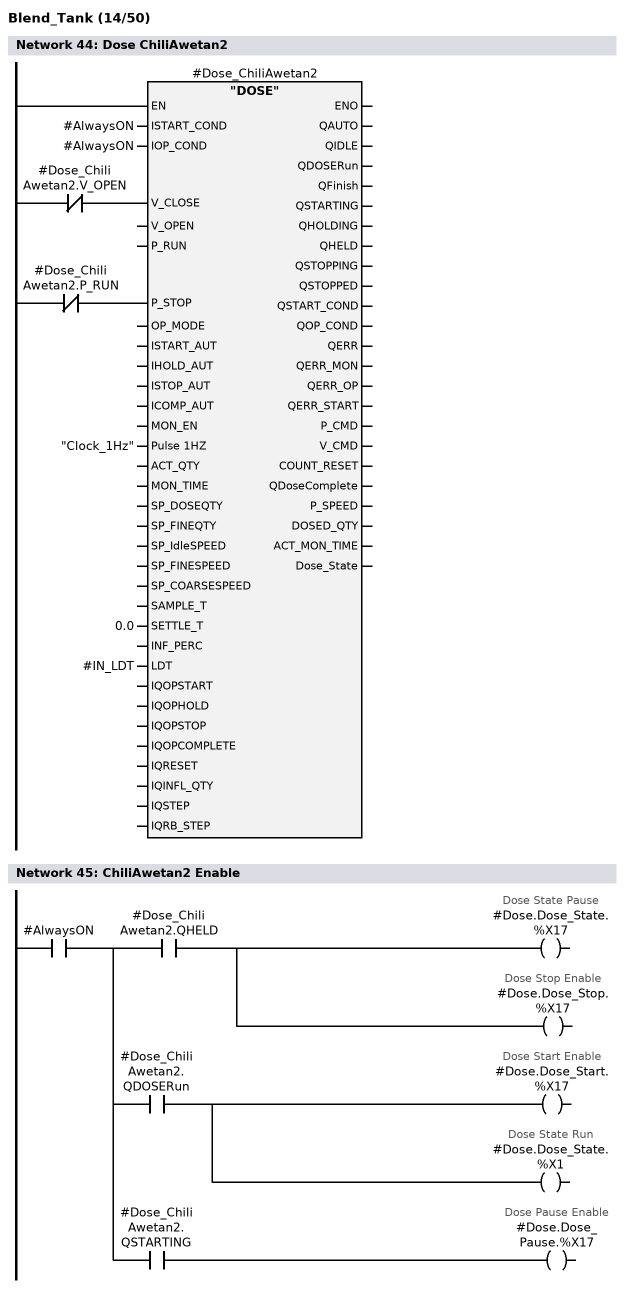
   RUNG wire#powerrail
      #Dose_ChiliAwetan2(V_CLOSE := wire#w1, P_STOP := wire#w2, ISTART_COND := #AlwaysON, IOP_COND := #AlwaysON, V_OPEN :=, P_RUN :=, OP_MODE :=, ISTART_AUT :=, IHOLD_AUT :=, ISTOP_AUT :=, ICOMP_AUT :=, MON_EN :=, "Pulse 1HZ" := "Clock_1Hz", ACT_QTY :=, MON_TIME :=, SP_DOSEQTY :=, SP_FINEQTY :=, SP_IdleSPEED :=, SP_FINESPEED :=, SP_COARSESPEED :=, SAMPLE_T :=, SETTLE_T := 0.0, INF_PERC :=, LDT := #IN_LDT, IQOPSTART :=, IQOPHOLD :=, IQOPSTOP :=, IQOPCOMPLETE :=, IQRESET :=, IQINFL_QTY :=, IQSTEP :=, IQRB_STEP :=, QAUTO =>, QIDLE =>, QDOSERun =>, QFinish =>, QSTARTING =>, QHOLDING =>, QHELD =>, QSTOPPING =>, QSTOPPED =>, QSTART_COND =>, QOP_COND =>, QERR =>, QERR_MON =>, QERR_OP =>, QERR_START =>, P_CMD =>, V_CMD =>, COUNT_RESET =>, QDoseComplete =>, P_SPEED =>, DOSED_QTY =>, ACT_MON_TIME =>, Dose_State =>)
   END_RUNG
   RUNG wire#powerrail
      I_Contact( #Dose_ChiliAwetan2.V_OPEN )
   END_RUNG wire#w1
   RUNG wire#powerrail
      I_Contact( #Dose_ChiliAwetan2.P_RUN )
   END_RUNG wire#w2
   // the same network as SCL:
   #Dose_ChiliAwetan2(ISTART_COND := #AlwaysON,   // "DOSE"
                      IOP_COND := #AlwaysON,
                      V_CLOSE := NOT #Dose_ChiliAwetan2.V_OPEN,
                      P_STOP := NOT #Dose_ChiliAwetan2.P_RUN,
                      "Pulse 1HZ" := "Clock_1Hz",
                      SETTLE_T := 0.0,
                      LDT := #IN_LDT);
END_REGION

REGION Network 45: ChiliAwetan2 Enable
   RUNG wire#powerrail
      Contact( #AlwaysON )
      wire#w1
      Contact( #Dose_ChiliAwetan2.QHELD )
      wire#w2
      Coil( #Dose.Dose_State.%X17 )   // Dose State Pause
   END_RUNG
   RUNG wire#w2
      Coil( #Dose.Dose_Stop.%X17 )   // Dose Stop Enable
   END_RUNG
   RUNG wire#w1
      Contact( #Dose_ChiliAwetan2.QDOSERun )
      wire#w3
      Coil( #Dose.Dose_Start.%X17 )   // Dose Start Enable
   END_RUNG
   RUNG wire#w3
      Coil( #Dose.Dose_State.%X1 )   // Dose State Run
   END_RUNG
   RUNG wire#w1
      Contact( #Dose_ChiliAwetan2.QSTARTING )
      Coil( #Dose.Dose_Pause.%X17 )   // Dose Pause Enable
   END_RUNG
   // the same network as SCL:
   #Dose.Dose_State.%X17 := #AlwaysON AND #Dose_ChiliAwetan2.QHELD;   // Dose State Pause
   #Dose.Dose_Stop.%X17 := #Dose.Dose_State.%X17;   // Dose Stop Enable
   #Dose.Dose_Start.%X17 := #AlwaysON AND #Dose_ChiliAwetan2.QDOSERun;   // Dose Start Enable
   #Dose.Dose_State.%X1 := #Dose.Dose_Start.%X17;   // Dose State Run
   #Dose.Dose_Pause.%X17 := #AlwaysON AND #Dose_ChiliAwetan2.QSTARTING;   // Dose Pause Enable
END_REGION

REGION Network 46: ChiliAwetan2 Header Req
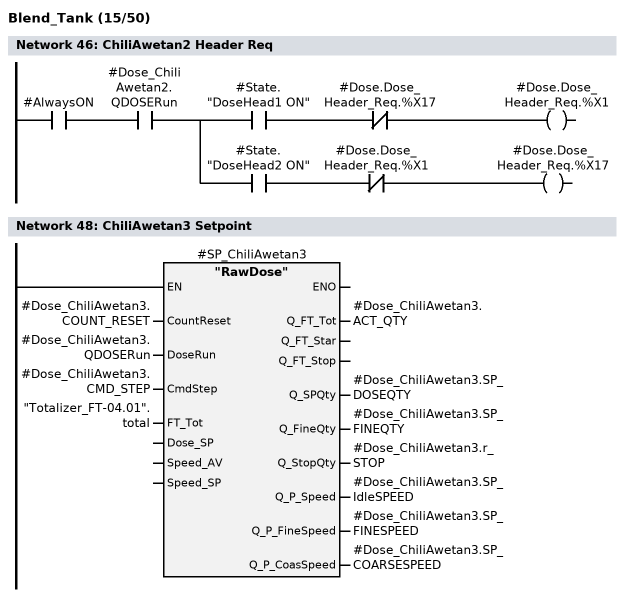
   RUNG wire#powerrail
      Contact( #AlwaysON )
      Contact( #Dose_ChiliAwetan2.QDOSERun )
      wire#w1
      Contact( #State."DoseHead1 ON" )
      I_Contact( #Dose.Dose_Header_Req.%X17 )
      Coil( #Dose.Dose_Header_Req.%X1 )
   END_RUNG
   RUNG wire#w1
      Contact( #State."DoseHead2 ON" )
      I_Contact( #Dose.Dose_Header_Req.%X1 )
      Coil( #Dose.Dose_Header_Req.%X17 )
   END_RUNG
   // the same network as SCL:
   #_w1 := #AlwaysON AND #Dose_ChiliAwetan2.QDOSERun;
   #Dose.Dose_Header_Req.%X1 := #_w1 AND #State."DoseHead1 ON" AND NOT #Dose.Dose_Header_Req.%X17;
   #Dose.Dose_Header_Req.%X17 := #_w1 AND #State."DoseHead2 ON" AND NOT #Dose.Dose_Header_Req.%X1;
END_REGION

REGION Network 48: ChiliAwetan3 Setpoint
   RUNG wire#powerrail
      #SP_ChiliAwetan3(CountReset := #Dose_ChiliAwetan3.COUNT_RESET, DoseRun := #Dose_ChiliAwetan3.QDOSERun, CmdStep := #Dose_ChiliAwetan3.CMD_STEP, FT_Tot := "Totalizer_FT-04.01".total, Dose_SP :=, Speed_AV :=, Speed_SP :=, Q_FT_Tot => #Dose_ChiliAwetan3.ACT_QTY, Q_FT_Star =>, Q_FT_Stop =>, Q_SPQty => #Dose_ChiliAwetan3.SP_DOSEQTY, Q_FineQty => #Dose_ChiliAwetan3.SP_FINEQTY, Q_StopQty => #Dose_ChiliAwetan3.r_STOP, Q_P_Speed => #Dose_ChiliAwetan3.SP_IdleSPEED, Q_P_FineSpeed => #Dose_ChiliAwetan3.SP_FINESPEED, Q_P_CoasSpeed => #Dose_ChiliAwetan3.SP_COARSESPEED)
   END_RUNG
   // the same network as SCL:
   #SP_ChiliAwetan3(CountReset := #Dose_ChiliAwetan3.COUNT_RESET,   // "RawDose"
                    DoseRun := #Dose_ChiliAwetan3.QDOSERun,
                    CmdStep := #Dose_ChiliAwetan3.CMD_STEP,
                    FT_Tot := "Totalizer_FT-04.01".total,
                    Q_FT_Tot => #Dose_ChiliAwetan3.ACT_QTY,
                    Q_SPQty => #Dose_ChiliAwetan3.SP_DOSEQTY,
                    Q_FineQty => #Dose_ChiliAwetan3.SP_FINEQTY,
                    Q_StopQty => #Dose_ChiliAwetan3.r_STOP,
                    Q_P_Speed => #Dose_ChiliAwetan3.SP_IdleSPEED,
                    Q_P_FineSpeed => #Dose_ChiliAwetan3.SP_FINESPEED,
                    Q_P_CoasSpeed => #Dose_ChiliAwetan3.SP_COARSESPEED);
END_REGION

REGION Network 49: Command Dose ChiliAwetan3
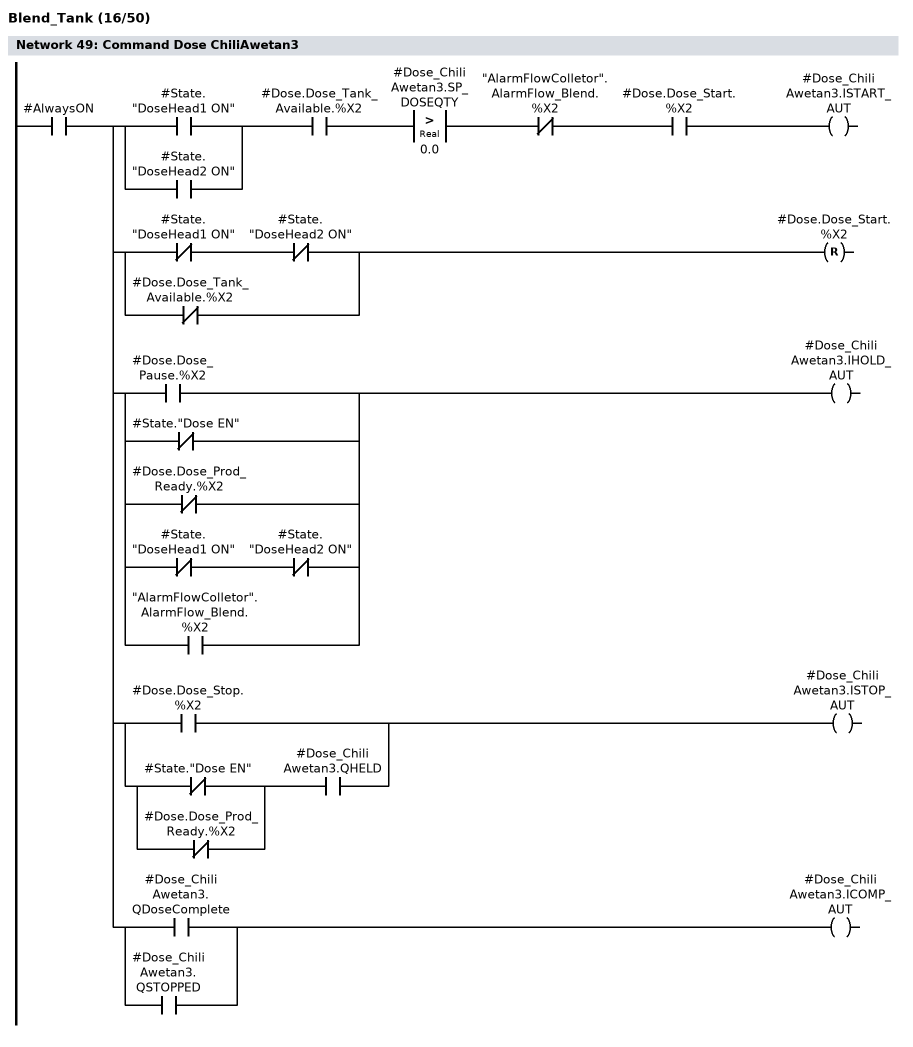
   RUNG wire#powerrail
      Contact( #AlwaysON )
      wire#w1
      Contact( #State."DoseHead1 ON" )
      wire#w2
      Contact( #Dose.Dose_Tank_Available.%X2 )
      { S7_Templates := "SrcType := Real" } GT_Contact(in1 := #Dose_ChiliAwetan3.SP_DOSEQTY, in2 := 0.0)
      I_Contact( "AlarmFlowColletor".AlarmFlow_Blend.%X2 )
      Contact( #Dose.Dose_Start.%X2 )
      Coil( #Dose_ChiliAwetan3.ISTART_AUT )
   END_RUNG
   RUNG wire#w1
      Contact( #State."DoseHead2 ON" )
   END_RUNG wire#w2
   RUNG wire#w1
      I_Contact( #State."DoseHead1 ON" )
      I_Contact( #State."DoseHead2 ON" )
      wire#w3
      R_Coil( #Dose.Dose_Start.%X2 )
   END_RUNG
   RUNG wire#w1
      I_Contact( #Dose.Dose_Tank_Available.%X2 )
   END_RUNG wire#w3
   RUNG wire#w1
      Contact( #Dose.Dose_Pause.%X2 )
      wire#w4
      Coil( #Dose_ChiliAwetan3.IHOLD_AUT )
   END_RUNG
   RUNG wire#w1
      I_Contact( #State."Dose EN" )
   END_RUNG wire#w4
   RUNG wire#w1
      I_Contact( #Dose.Dose_Prod_Ready.%X2 )
   END_RUNG wire#w4
   RUNG wire#w1
      I_Contact( #State."DoseHead1 ON" )
      I_Contact( #State."DoseHead2 ON" )
   END_RUNG wire#w4
   RUNG wire#w1
      Contact( "AlarmFlowColletor".AlarmFlow_Blend.%X2 )
   END_RUNG wire#w4
   RUNG wire#w1
      Contact( #Dose.Dose_Stop.%X2 )
      wire#w5
      Coil( #Dose_ChiliAwetan3.ISTOP_AUT )
   END_RUNG
   RUNG wire#w1
      I_Contact( #State."Dose EN" )
      wire#w6
      Contact( #Dose_ChiliAwetan3.QHELD )
   END_RUNG wire#w5
   RUNG wire#w1
      I_Contact( #Dose.Dose_Prod_Ready.%X2 )
   END_RUNG wire#w6
   RUNG wire#w1
      Contact( #Dose_ChiliAwetan3.QDoseComplete )
      wire#w7
      Coil( #Dose_ChiliAwetan3.ICOMP_AUT )
   END_RUNG
   RUNG wire#w1
      Contact( #Dose_ChiliAwetan3.QSTOPPED )
   END_RUNG wire#w7
   // the same network as SCL:
   #Dose_ChiliAwetan3.ISTART_AUT := #AlwaysON AND (#State."DoseHead1 ON" OR #State."DoseHead2 ON") AND #Dose.Dose_Tank_Available.%X2 AND (#Dose_ChiliAwetan3.SP_DOSEQTY > 0.0) AND NOT "AlarmFlowColletor".AlarmFlow_Blend.%X2 AND #Dose.Dose_Start.%X2;
   IF #AlwaysON AND ((NOT #State."DoseHead1 ON" AND NOT #State."DoseHead2 ON") OR NOT #Dose.Dose_Tank_Available.%X2) THEN
       #Dose.Dose_Start.%X2 := FALSE;
   END_IF;
   #Dose_ChiliAwetan3.IHOLD_AUT := #AlwaysON AND (#Dose.Dose_Pause.%X2 OR NOT #State."Dose EN" OR NOT #Dose.Dose_Prod_Ready.%X2 OR (NOT #State."DoseHead1 ON" AND NOT #State."DoseHead2 ON") OR "AlarmFlowColletor".AlarmFlow_Blend.%X2);
   #Dose_ChiliAwetan3.ISTOP_AUT := #AlwaysON AND (#Dose.Dose_Stop.%X2 OR ((NOT #State."Dose EN" OR NOT #Dose.Dose_Prod_Ready.%X2) AND #Dose_ChiliAwetan3.QHELD));
   #Dose_ChiliAwetan3.ICOMP_AUT := #AlwaysON AND (#Dose_ChiliAwetan3.QDoseComplete OR #Dose_ChiliAwetan3.QSTOPPED);
END_REGION

REGION Network 50: Dose ChiliAwetan3
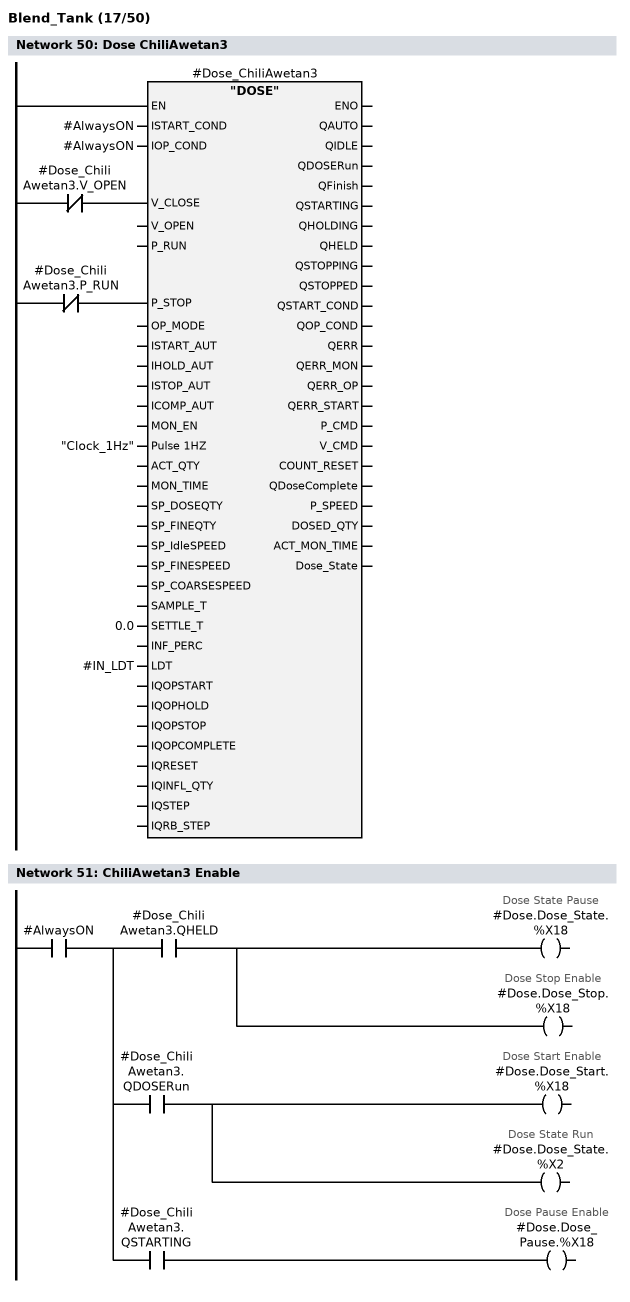
   RUNG wire#powerrail
      #Dose_ChiliAwetan3(V_CLOSE := wire#w1, P_STOP := wire#w2, ISTART_COND := #AlwaysON, IOP_COND := #AlwaysON, V_OPEN :=, P_RUN :=, OP_MODE :=, ISTART_AUT :=, IHOLD_AUT :=, ISTOP_AUT :=, ICOMP_AUT :=, MON_EN :=, "Pulse 1HZ" := "Clock_1Hz", ACT_QTY :=, MON_TIME :=, SP_DOSEQTY :=, SP_FINEQTY :=, SP_IdleSPEED :=, SP_FINESPEED :=, SP_COARSESPEED :=, SAMPLE_T :=, SETTLE_T := 0.0, INF_PERC :=, LDT := #IN_LDT, IQOPSTART :=, IQOPHOLD :=, IQOPSTOP :=, IQOPCOMPLETE :=, IQRESET :=, IQINFL_QTY :=, IQSTEP :=, IQRB_STEP :=, QAUTO =>, QIDLE =>, QDOSERun =>, QFinish =>, QSTARTING =>, QHOLDING =>, QHELD =>, QSTOPPING =>, QSTOPPED =>, QSTART_COND =>, QOP_COND =>, QERR =>, QERR_MON =>, QERR_OP =>, QERR_START =>, P_CMD =>, V_CMD =>, COUNT_RESET =>, QDoseComplete =>, P_SPEED =>, DOSED_QTY =>, ACT_MON_TIME =>, Dose_State =>)
   END_RUNG
   RUNG wire#powerrail
      I_Contact( #Dose_ChiliAwetan3.V_OPEN )
   END_RUNG wire#w1
   RUNG wire#powerrail
      I_Contact( #Dose_ChiliAwetan3.P_RUN )
   END_RUNG wire#w2
   // the same network as SCL:
   #Dose_ChiliAwetan3(ISTART_COND := #AlwaysON,   // "DOSE"
                      IOP_COND := #AlwaysON,
                      V_CLOSE := NOT #Dose_ChiliAwetan3.V_OPEN,
                      P_STOP := NOT #Dose_ChiliAwetan3.P_RUN,
                      "Pulse 1HZ" := "Clock_1Hz",
                      SETTLE_T := 0.0,
                      LDT := #IN_LDT);
END_REGION

REGION Network 51: ChiliAwetan3 Enable
   RUNG wire#powerrail
      Contact( #AlwaysON )
      wire#w1
      Contact( #Dose_ChiliAwetan3.QHELD )
      wire#w2
      Coil( #Dose.Dose_State.%X18 )   // Dose State Pause
   END_RUNG
   RUNG wire#w2
      Coil( #Dose.Dose_Stop.%X18 )   // Dose Stop Enable
   END_RUNG
   RUNG wire#w1
      Contact( #Dose_ChiliAwetan3.QDOSERun )
      wire#w3
      Coil( #Dose.Dose_Start.%X18 )   // Dose Start Enable
   END_RUNG
   RUNG wire#w3
      Coil( #Dose.Dose_State.%X2 )   // Dose State Run
   END_RUNG
   RUNG wire#w1
      Contact( #Dose_ChiliAwetan3.QSTARTING )
      Coil( #Dose.Dose_Pause.%X18 )   // Dose Pause Enable
   END_RUNG
   // the same network as SCL:
   #Dose.Dose_State.%X18 := #AlwaysON AND #Dose_ChiliAwetan3.QHELD;   // Dose State Pause
   #Dose.Dose_Stop.%X18 := #Dose.Dose_State.%X18;   // Dose Stop Enable
   #Dose.Dose_Start.%X18 := #AlwaysON AND #Dose_ChiliAwetan3.QDOSERun;   // Dose Start Enable
   #Dose.Dose_State.%X2 := #Dose.Dose_Start.%X18;   // Dose State Run
   #Dose.Dose_Pause.%X18 := #AlwaysON AND #Dose_ChiliAwetan3.QSTARTING;   // Dose Pause Enable
END_REGION

REGION Network 52: ChiliAwetan3 Header Req
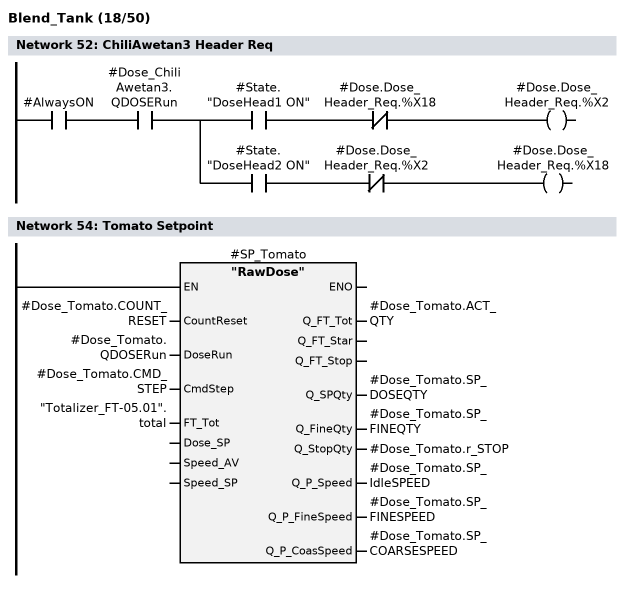
   RUNG wire#powerrail
      Contact( #AlwaysON )
      Contact( #Dose_ChiliAwetan3.QDOSERun )
      wire#w1
      Contact( #State."DoseHead1 ON" )
      I_Contact( #Dose.Dose_Header_Req.%X18 )
      Coil( #Dose.Dose_Header_Req.%X2 )
   END_RUNG
   RUNG wire#w1
      Contact( #State."DoseHead2 ON" )
      I_Contact( #Dose.Dose_Header_Req.%X2 )
      Coil( #Dose.Dose_Header_Req.%X18 )
   END_RUNG
   // the same network as SCL:
   #_w1 := #AlwaysON AND #Dose_ChiliAwetan3.QDOSERun;
   #Dose.Dose_Header_Req.%X2 := #_w1 AND #State."DoseHead1 ON" AND NOT #Dose.Dose_Header_Req.%X18;
   #Dose.Dose_Header_Req.%X18 := #_w1 AND #State."DoseHead2 ON" AND NOT #Dose.Dose_Header_Req.%X2;
END_REGION

REGION Network 54: Tomato Setpoint
   RUNG wire#powerrail
      #SP_Tomato(CountReset := #Dose_Tomato.COUNT_RESET, DoseRun := #Dose_Tomato.QDOSERun, CmdStep := #Dose_Tomato.CMD_STEP, FT_Tot := "Totalizer_FT-05.01".total, Dose_SP :=, Speed_AV :=, Speed_SP :=, Q_FT_Tot => #Dose_Tomato.ACT_QTY, Q_FT_Star =>, Q_FT_Stop =>, Q_SPQty => #Dose_Tomato.SP_DOSEQTY, Q_FineQty => #Dose_Tomato.SP_FINEQTY, Q_StopQty => #Dose_Tomato.r_STOP, Q_P_Speed => #Dose_Tomato.SP_IdleSPEED, Q_P_FineSpeed => #Dose_Tomato.SP_FINESPEED, Q_P_CoasSpeed => #Dose_Tomato.SP_COARSESPEED)
   END_RUNG
   // the same network as SCL:
   #SP_Tomato(CountReset := #Dose_Tomato.COUNT_RESET,   // "RawDose"
              DoseRun := #Dose_Tomato.QDOSERun,
              CmdStep := #Dose_Tomato.CMD_STEP,
              FT_Tot := "Totalizer_FT-05.01".total,
              Q_FT_Tot => #Dose_Tomato.ACT_QTY,
              Q_SPQty => #Dose_Tomato.SP_DOSEQTY,
              Q_FineQty => #Dose_Tomato.SP_FINEQTY,
              Q_StopQty => #Dose_Tomato.r_STOP,
              Q_P_Speed => #Dose_Tomato.SP_IdleSPEED,
              Q_P_FineSpeed => #Dose_Tomato.SP_FINESPEED,
              Q_P_CoasSpeed => #Dose_Tomato.SP_COARSESPEED);
END_REGION

REGION Network 55: Command Dose Tomato
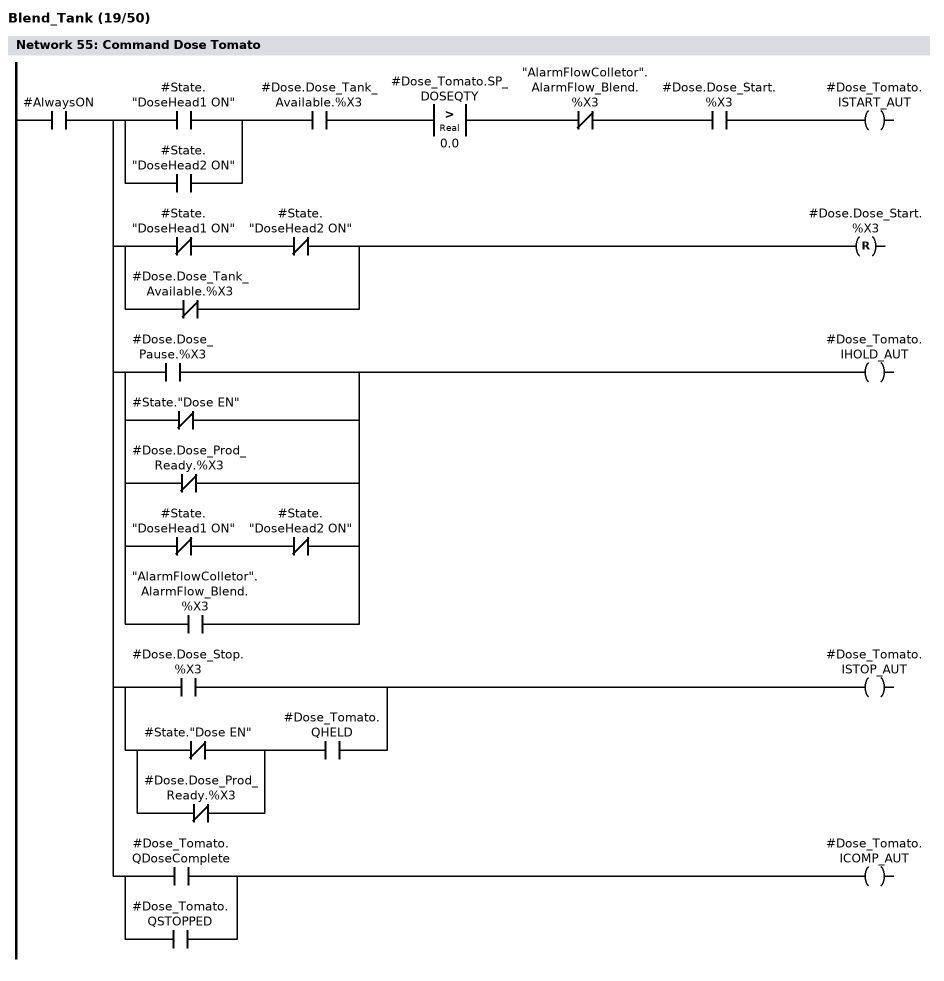
   RUNG wire#powerrail
      Contact( #AlwaysON )
      wire#w1
      Contact( #State."DoseHead1 ON" )
      wire#w2
      Contact( #Dose.Dose_Tank_Available.%X3 )
      { S7_Templates := "SrcType := Real" } GT_Contact(in1 := #Dose_Tomato.SP_DOSEQTY, in2 := 0.0)
      I_Contact( "AlarmFlowColletor".AlarmFlow_Blend.%X3 )
      Contact( #Dose.Dose_Start.%X3 )
      Coil( #Dose_Tomato.ISTART_AUT )
   END_RUNG
   RUNG wire#w1
      Contact( #State."DoseHead2 ON" )
   END_RUNG wire#w2
   RUNG wire#w1
      I_Contact( #State."DoseHead1 ON" )
      I_Contact( #State."DoseHead2 ON" )
      wire#w3
      R_Coil( #Dose.Dose_Start.%X3 )
   END_RUNG
   RUNG wire#w1
      I_Contact( #Dose.Dose_Tank_Available.%X3 )
   END_RUNG wire#w3
   RUNG wire#w1
      Contact( #Dose.Dose_Pause.%X3 )
      wire#w4
      Coil( #Dose_Tomato.IHOLD_AUT )
   END_RUNG
   RUNG wire#w1
      I_Contact( #State."Dose EN" )
   END_RUNG wire#w4
   RUNG wire#w1
      I_Contact( #Dose.Dose_Prod_Ready.%X3 )
   END_RUNG wire#w4
   RUNG wire#w1
      I_Contact( #State."DoseHead1 ON" )
      I_Contact( #State."DoseHead2 ON" )
   END_RUNG wire#w4
   RUNG wire#w1
      Contact( "AlarmFlowColletor".AlarmFlow_Blend.%X3 )
   END_RUNG wire#w4
   RUNG wire#w1
      Contact( #Dose.Dose_Stop.%X3 )
      wire#w5
      Coil( #Dose_Tomato.ISTOP_AUT )
   END_RUNG
   RUNG wire#w1
      I_Contact( #State."Dose EN" )
      wire#w6
      Contact( #Dose_Tomato.QHELD )
   END_RUNG wire#w5
   RUNG wire#w1
      I_Contact( #Dose.Dose_Prod_Ready.%X3 )
   END_RUNG wire#w6
   RUNG wire#w1
      Contact( #Dose_Tomato.QDoseComplete )
      wire#w7
      Coil( #Dose_Tomato.ICOMP_AUT )
   END_RUNG
   RUNG wire#w1
      Contact( #Dose_Tomato.QSTOPPED )
   END_RUNG wire#w7
   // the same network as SCL:
   #Dose_Tomato.ISTART_AUT := #AlwaysON AND (#State."DoseHead1 ON" OR #State."DoseHead2 ON") AND #Dose.Dose_Tank_Available.%X3 AND (#Dose_Tomato.SP_DOSEQTY > 0.0) AND NOT "AlarmFlowColletor".AlarmFlow_Blend.%X3 AND #Dose.Dose_Start.%X3;
   IF #AlwaysON AND ((NOT #State."DoseHead1 ON" AND NOT #State."DoseHead2 ON") OR NOT #Dose.Dose_Tank_Available.%X3) THEN
       #Dose.Dose_Start.%X3 := FALSE;
   END_IF;
   #Dose_Tomato.IHOLD_AUT := #AlwaysON AND (#Dose.Dose_Pause.%X3 OR NOT #State."Dose EN" OR NOT #Dose.Dose_Prod_Ready.%X3 OR (NOT #State."DoseHead1 ON" AND NOT #State."DoseHead2 ON") OR "AlarmFlowColletor".AlarmFlow_Blend.%X3);
   #Dose_Tomato.ISTOP_AUT := #AlwaysON AND (#Dose.Dose_Stop.%X3 OR ((NOT #State."Dose EN" OR NOT #Dose.Dose_Prod_Ready.%X3) AND #Dose_Tomato.QHELD));
   #Dose_Tomato.ICOMP_AUT := #AlwaysON AND (#Dose_Tomato.QDoseComplete OR #Dose_Tomato.QSTOPPED);
END_REGION

REGION Network 56: Dose Tomato
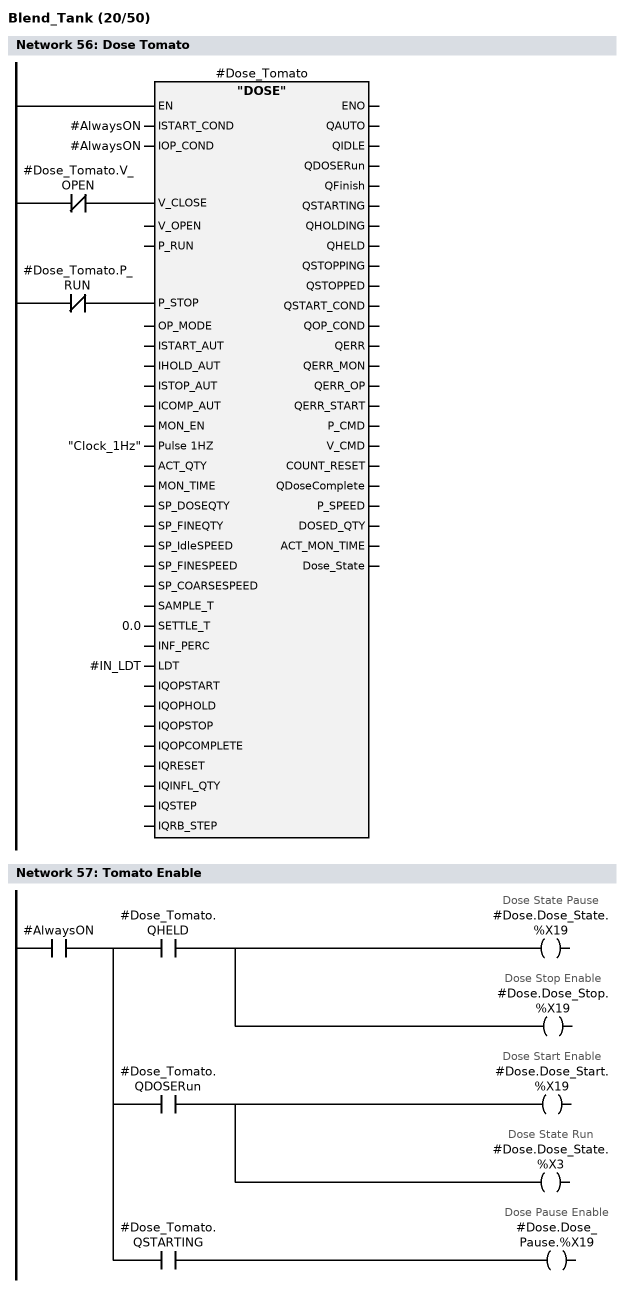
   RUNG wire#powerrail
      #Dose_Tomato(V_CLOSE := wire#w1, P_STOP := wire#w2, ISTART_COND := #AlwaysON, IOP_COND := #AlwaysON, V_OPEN :=, P_RUN :=, OP_MODE :=, ISTART_AUT :=, IHOLD_AUT :=, ISTOP_AUT :=, ICOMP_AUT :=, MON_EN :=, "Pulse 1HZ" := "Clock_1Hz", ACT_QTY :=, MON_TIME :=, SP_DOSEQTY :=, SP_FINEQTY :=, SP_IdleSPEED :=, SP_FINESPEED :=, SP_COARSESPEED :=, SAMPLE_T :=, SETTLE_T := 0.0, INF_PERC :=, LDT := #IN_LDT, IQOPSTART :=, IQOPHOLD :=, IQOPSTOP :=, IQOPCOMPLETE :=, IQRESET :=, IQINFL_QTY :=, IQSTEP :=, IQRB_STEP :=, QAUTO =>, QIDLE =>, QDOSERun =>, QFinish =>, QSTARTING =>, QHOLDING =>, QHELD =>, QSTOPPING =>, QSTOPPED =>, QSTART_COND =>, QOP_COND =>, QERR =>, QERR_MON =>, QERR_OP =>, QERR_START =>, P_CMD =>, V_CMD =>, COUNT_RESET =>, QDoseComplete =>, P_SPEED =>, DOSED_QTY =>, ACT_MON_TIME =>, Dose_State =>)
   END_RUNG
   RUNG wire#powerrail
      I_Contact( #Dose_Tomato.V_OPEN )
   END_RUNG wire#w1
   RUNG wire#powerrail
      I_Contact( #Dose_Tomato.P_RUN )
   END_RUNG wire#w2
   // the same network as SCL:
   #Dose_Tomato(ISTART_COND := #AlwaysON,   // "DOSE"
                IOP_COND := #AlwaysON,
                V_CLOSE := NOT #Dose_Tomato.V_OPEN,
                P_STOP := NOT #Dose_Tomato.P_RUN,
                "Pulse 1HZ" := "Clock_1Hz",
                SETTLE_T := 0.0,
                LDT := #IN_LDT);
END_REGION

REGION Network 57: Tomato Enable
   RUNG wire#powerrail
      Contact( #AlwaysON )
      wire#w1
      Contact( #Dose_Tomato.QHELD )
      wire#w2
      Coil( #Dose.Dose_State.%X19 )   // Dose State Pause
   END_RUNG
   RUNG wire#w2
      Coil( #Dose.Dose_Stop.%X19 )   // Dose Stop Enable
   END_RUNG
   RUNG wire#w1
      Contact( #Dose_Tomato.QDOSERun )
      wire#w3
      Coil( #Dose.Dose_Start.%X19 )   // Dose Start Enable
   END_RUNG
   RUNG wire#w3
      Coil( #Dose.Dose_State.%X3 )   // Dose State Run
   END_RUNG
   RUNG wire#w1
      Contact( #Dose_Tomato.QSTARTING )
      Coil( #Dose.Dose_Pause.%X19 )   // Dose Pause Enable
   END_RUNG
   // the same network as SCL:
   #Dose.Dose_State.%X19 := #AlwaysON AND #Dose_Tomato.QHELD;   // Dose State Pause
   #Dose.Dose_Stop.%X19 := #Dose.Dose_State.%X19;   // Dose Stop Enable
   #Dose.Dose_Start.%X19 := #AlwaysON AND #Dose_Tomato.QDOSERun;   // Dose Start Enable
   #Dose.Dose_State.%X3 := #Dose.Dose_Start.%X19;   // Dose State Run
   #Dose.Dose_Pause.%X19 := #AlwaysON AND #Dose_Tomato.QSTARTING;   // Dose Pause Enable
END_REGION

REGION Network 58: Tomato Header Req
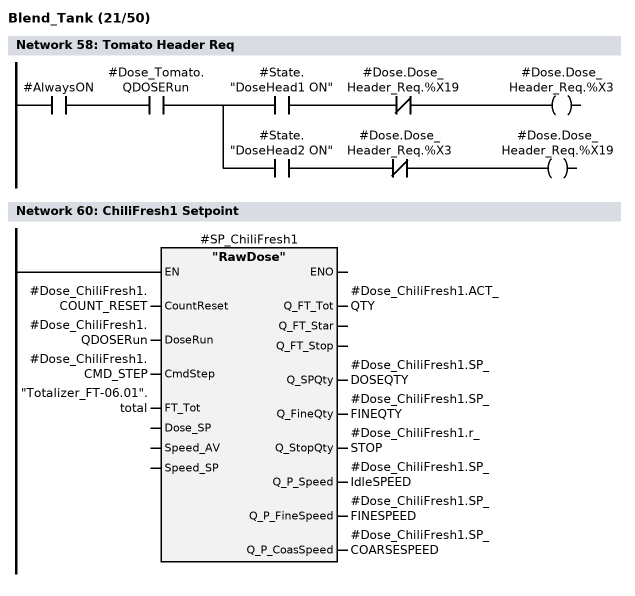
   RUNG wire#powerrail
      Contact( #AlwaysON )
      Contact( #Dose_Tomato.QDOSERun )
      wire#w1
      Contact( #State."DoseHead1 ON" )
      I_Contact( #Dose.Dose_Header_Req.%X19 )
      Coil( #Dose.Dose_Header_Req.%X3 )
   END_RUNG
   RUNG wire#w1
      Contact( #State."DoseHead2 ON" )
      I_Contact( #Dose.Dose_Header_Req.%X3 )
      Coil( #Dose.Dose_Header_Req.%X19 )
   END_RUNG
   // the same network as SCL:
   #_w1 := #AlwaysON AND #Dose_Tomato.QDOSERun;
   #Dose.Dose_Header_Req.%X3 := #_w1 AND #State."DoseHead1 ON" AND NOT #Dose.Dose_Header_Req.%X19;
   #Dose.Dose_Header_Req.%X19 := #_w1 AND #State."DoseHead2 ON" AND NOT #Dose.Dose_Header_Req.%X3;
END_REGION

REGION Network 60: ChiliFresh1 Setpoint
   RUNG wire#powerrail
      #SP_ChiliFresh1(CountReset := #Dose_ChiliFresh1.COUNT_RESET, DoseRun := #Dose_ChiliFresh1.QDOSERun, CmdStep := #Dose_ChiliFresh1.CMD_STEP, FT_Tot := "Totalizer_FT-06.01".total, Dose_SP :=, Speed_AV :=, Speed_SP :=, Q_FT_Tot => #Dose_ChiliFresh1.ACT_QTY, Q_FT_Star =>, Q_FT_Stop =>, Q_SPQty => #Dose_ChiliFresh1.SP_DOSEQTY, Q_FineQty => #Dose_ChiliFresh1.SP_FINEQTY, Q_StopQty => #Dose_ChiliFresh1.r_STOP, Q_P_Speed => #Dose_ChiliFresh1.SP_IdleSPEED, Q_P_FineSpeed => #Dose_ChiliFresh1.SP_FINESPEED, Q_P_CoasSpeed => #Dose_ChiliFresh1.SP_COARSESPEED)
   END_RUNG
   // the same network as SCL:
   #SP_ChiliFresh1(CountReset := #Dose_ChiliFresh1.COUNT_RESET,   // "RawDose"
                   DoseRun := #Dose_ChiliFresh1.QDOSERun,
                   CmdStep := #Dose_ChiliFresh1.CMD_STEP,
                   FT_Tot := "Totalizer_FT-06.01".total,
                   Q_FT_Tot => #Dose_ChiliFresh1.ACT_QTY,
                   Q_SPQty => #Dose_ChiliFresh1.SP_DOSEQTY,
                   Q_FineQty => #Dose_ChiliFresh1.SP_FINEQTY,
                   Q_StopQty => #Dose_ChiliFresh1.r_STOP,
                   Q_P_Speed => #Dose_ChiliFresh1.SP_IdleSPEED,
                   Q_P_FineSpeed => #Dose_ChiliFresh1.SP_FINESPEED,
                   Q_P_CoasSpeed => #Dose_ChiliFresh1.SP_COARSESPEED);
END_REGION

REGION Network 61: Command Dose ChiliFresh1
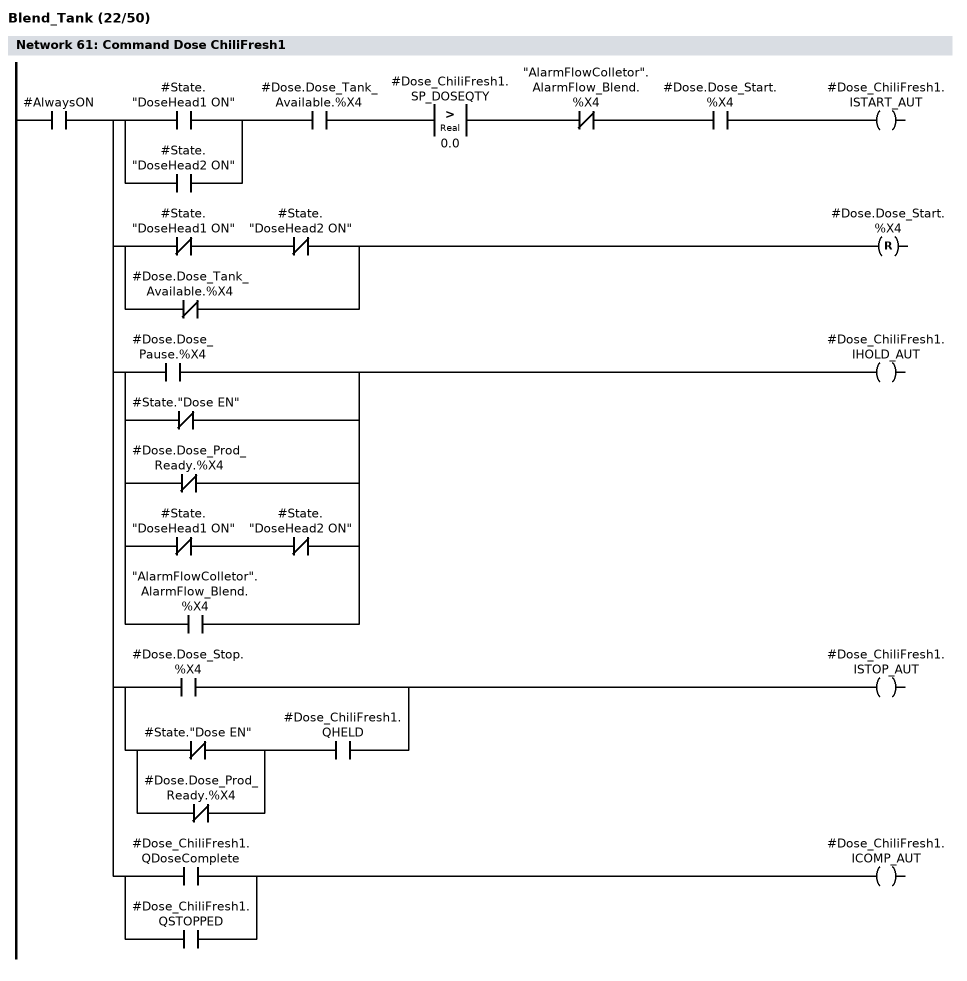
   RUNG wire#powerrail
      Contact( #AlwaysON )
      wire#w1
      Contact( #State."DoseHead1 ON" )
      wire#w2
      Contact( #Dose.Dose_Tank_Available.%X4 )
      { S7_Templates := "SrcType := Real" } GT_Contact(in1 := #Dose_ChiliFresh1.SP_DOSEQTY, in2 := 0.0)
      I_Contact( "AlarmFlowColletor".AlarmFlow_Blend.%X4 )
      Contact( #Dose.Dose_Start.%X4 )
      Coil( #Dose_ChiliFresh1.ISTART_AUT )
   END_RUNG
   RUNG wire#w1
      Contact( #State."DoseHead2 ON" )
   END_RUNG wire#w2
   RUNG wire#w1
      I_Contact( #State."DoseHead1 ON" )
      I_Contact( #State."DoseHead2 ON" )
      wire#w3
      R_Coil( #Dose.Dose_Start.%X4 )
   END_RUNG
   RUNG wire#w1
      I_Contact( #Dose.Dose_Tank_Available.%X4 )
   END_RUNG wire#w3
   RUNG wire#w1
      Contact( #Dose.Dose_Pause.%X4 )
      wire#w4
      Coil( #Dose_ChiliFresh1.IHOLD_AUT )
   END_RUNG
   RUNG wire#w1
      I_Contact( #State."Dose EN" )
   END_RUNG wire#w4
   RUNG wire#w1
      I_Contact( #Dose.Dose_Prod_Ready.%X4 )
   END_RUNG wire#w4
   RUNG wire#w1
      I_Contact( #State."DoseHead1 ON" )
      I_Contact( #State."DoseHead2 ON" )
   END_RUNG wire#w4
   RUNG wire#w1
      Contact( "AlarmFlowColletor".AlarmFlow_Blend.%X4 )
   END_RUNG wire#w4
   RUNG wire#w1
      Contact( #Dose.Dose_Stop.%X4 )
      wire#w5
      Coil( #Dose_ChiliFresh1.ISTOP_AUT )
   END_RUNG
   RUNG wire#w1
      I_Contact( #State."Dose EN" )
      wire#w6
      Contact( #Dose_ChiliFresh1.QHELD )
   END_RUNG wire#w5
   RUNG wire#w1
      I_Contact( #Dose.Dose_Prod_Ready.%X4 )
   END_RUNG wire#w6
   RUNG wire#w1
      Contact( #Dose_ChiliFresh1.QDoseComplete )
      wire#w7
      Coil( #Dose_ChiliFresh1.ICOMP_AUT )
   END_RUNG
   RUNG wire#w1
      Contact( #Dose_ChiliFresh1.QSTOPPED )
   END_RUNG wire#w7
   // the same network as SCL:
   #Dose_ChiliFresh1.ISTART_AUT := #AlwaysON AND (#State."DoseHead1 ON" OR #State."DoseHead2 ON") AND #Dose.Dose_Tank_Available.%X4 AND (#Dose_ChiliFresh1.SP_DOSEQTY > 0.0) AND NOT "AlarmFlowColletor".AlarmFlow_Blend.%X4 AND #Dose.Dose_Start.%X4;
   IF #AlwaysON AND ((NOT #State."DoseHead1 ON" AND NOT #State."DoseHead2 ON") OR NOT #Dose.Dose_Tank_Available.%X4) THEN
       #Dose.Dose_Start.%X4 := FALSE;
   END_IF;
   #Dose_ChiliFresh1.IHOLD_AUT := #AlwaysON AND (#Dose.Dose_Pause.%X4 OR NOT #State."Dose EN" OR NOT #Dose.Dose_Prod_Ready.%X4 OR (NOT #State."DoseHead1 ON" AND NOT #State."DoseHead2 ON") OR "AlarmFlowColletor".AlarmFlow_Blend.%X4);
   #Dose_ChiliFresh1.ISTOP_AUT := #AlwaysON AND (#Dose.Dose_Stop.%X4 OR ((NOT #State."Dose EN" OR NOT #Dose.Dose_Prod_Ready.%X4) AND #Dose_ChiliFresh1.QHELD));
   #Dose_ChiliFresh1.ICOMP_AUT := #AlwaysON AND (#Dose_ChiliFresh1.QDoseComplete OR #Dose_ChiliFresh1.QSTOPPED);
END_REGION

REGION Network 62: Dose ChiliFresh1
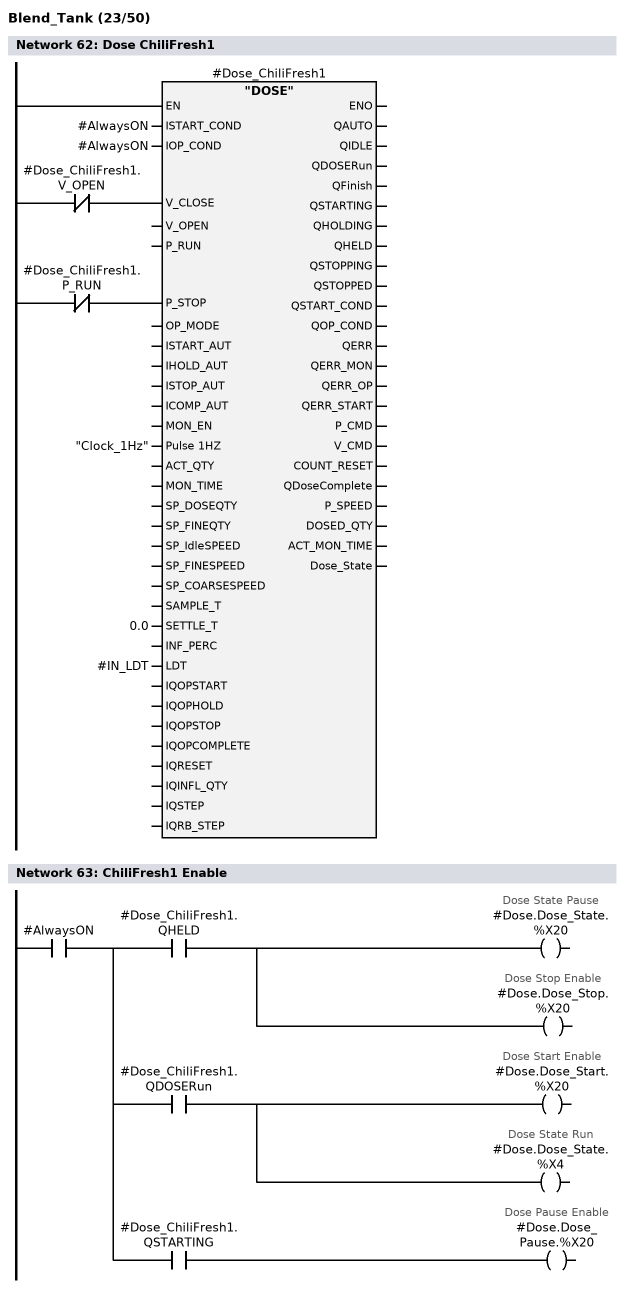
   RUNG wire#powerrail
      #Dose_ChiliFresh1(V_CLOSE := wire#w1, P_STOP := wire#w2, ISTART_COND := #AlwaysON, IOP_COND := #AlwaysON, V_OPEN :=, P_RUN :=, OP_MODE :=, ISTART_AUT :=, IHOLD_AUT :=, ISTOP_AUT :=, ICOMP_AUT :=, MON_EN :=, "Pulse 1HZ" := "Clock_1Hz", ACT_QTY :=, MON_TIME :=, SP_DOSEQTY :=, SP_FINEQTY :=, SP_IdleSPEED :=, SP_FINESPEED :=, SP_COARSESPEED :=, SAMPLE_T :=, SETTLE_T := 0.0, INF_PERC :=, LDT := #IN_LDT, IQOPSTART :=, IQOPHOLD :=, IQOPSTOP :=, IQOPCOMPLETE :=, IQRESET :=, IQINFL_QTY :=, IQSTEP :=, IQRB_STEP :=, QAUTO =>, QIDLE =>, QDOSERun =>, QFinish =>, QSTARTING =>, QHOLDING =>, QHELD =>, QSTOPPING =>, QSTOPPED =>, QSTART_COND =>, QOP_COND =>, QERR =>, QERR_MON =>, QERR_OP =>, QERR_START =>, P_CMD =>, V_CMD =>, COUNT_RESET =>, QDoseComplete =>, P_SPEED =>, DOSED_QTY =>, ACT_MON_TIME =>, Dose_State =>)
   END_RUNG
   RUNG wire#powerrail
      I_Contact( #Dose_ChiliFresh1.V_OPEN )
   END_RUNG wire#w1
   RUNG wire#powerrail
      I_Contact( #Dose_ChiliFresh1.P_RUN )
   END_RUNG wire#w2
   // the same network as SCL:
   #Dose_ChiliFresh1(ISTART_COND := #AlwaysON,   // "DOSE"
                     IOP_COND := #AlwaysON,
                     V_CLOSE := NOT #Dose_ChiliFresh1.V_OPEN,
                     P_STOP := NOT #Dose_ChiliFresh1.P_RUN,
                     "Pulse 1HZ" := "Clock_1Hz",
                     SETTLE_T := 0.0,
                     LDT := #IN_LDT);
END_REGION

REGION Network 63: ChiliFresh1 Enable
   RUNG wire#powerrail
      Contact( #AlwaysON )
      wire#w1
      Contact( #Dose_ChiliFresh1.QHELD )
      wire#w2
      Coil( #Dose.Dose_State.%X20 )   // Dose State Pause
   END_RUNG
   RUNG wire#w2
      Coil( #Dose.Dose_Stop.%X20 )   // Dose Stop Enable
   END_RUNG
   RUNG wire#w1
      Contact( #Dose_ChiliFresh1.QDOSERun )
      wire#w3
      Coil( #Dose.Dose_Start.%X20 )   // Dose Start Enable
   END_RUNG
   RUNG wire#w3
      Coil( #Dose.Dose_State.%X4 )   // Dose State Run
   END_RUNG
   RUNG wire#w1
      Contact( #Dose_ChiliFresh1.QSTARTING )
      Coil( #Dose.Dose_Pause.%X20 )   // Dose Pause Enable
   END_RUNG
   // the same network as SCL:
   #Dose.Dose_State.%X20 := #AlwaysON AND #Dose_ChiliFresh1.QHELD;   // Dose State Pause
   #Dose.Dose_Stop.%X20 := #Dose.Dose_State.%X20;   // Dose Stop Enable
   #Dose.Dose_Start.%X20 := #AlwaysON AND #Dose_ChiliFresh1.QDOSERun;   // Dose Start Enable
   #Dose.Dose_State.%X4 := #Dose.Dose_Start.%X20;   // Dose State Run
   #Dose.Dose_Pause.%X20 := #AlwaysON AND #Dose_ChiliFresh1.QSTARTING;   // Dose Pause Enable
END_REGION

REGION Network 64: ChiliFresh1 Header Req
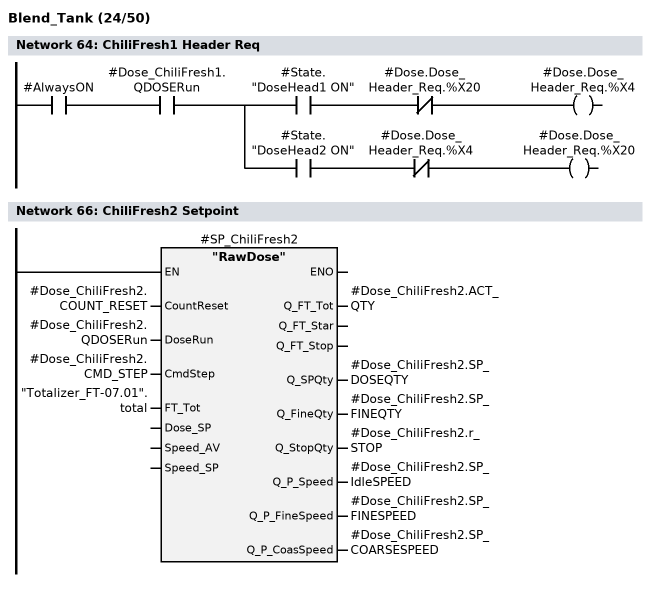
   RUNG wire#powerrail
      Contact( #AlwaysON )
      Contact( #Dose_ChiliFresh1.QDOSERun )
      wire#w1
      Contact( #State."DoseHead1 ON" )
      I_Contact( #Dose.Dose_Header_Req.%X20 )
      Coil( #Dose.Dose_Header_Req.%X4 )
   END_RUNG
   RUNG wire#w1
      Contact( #State."DoseHead2 ON" )
      I_Contact( #Dose.Dose_Header_Req.%X4 )
      Coil( #Dose.Dose_Header_Req.%X20 )
   END_RUNG
   // the same network as SCL:
   #_w1 := #AlwaysON AND #Dose_ChiliFresh1.QDOSERun;
   #Dose.Dose_Header_Req.%X4 := #_w1 AND #State."DoseHead1 ON" AND NOT #Dose.Dose_Header_Req.%X20;
   #Dose.Dose_Header_Req.%X20 := #_w1 AND #State."DoseHead2 ON" AND NOT #Dose.Dose_Header_Req.%X4;
END_REGION

REGION Network 66: ChiliFresh2 Setpoint
   RUNG wire#powerrail
      #SP_ChiliFresh2(CountReset := #Dose_ChiliFresh2.COUNT_RESET, DoseRun := #Dose_ChiliFresh2.QDOSERun, CmdStep := #Dose_ChiliFresh2.CMD_STEP, FT_Tot := "Totalizer_FT-07.01".total, Dose_SP :=, Speed_AV :=, Speed_SP :=, Q_FT_Tot => #Dose_ChiliFresh2.ACT_QTY, Q_FT_Star =>, Q_FT_Stop =>, Q_SPQty => #Dose_ChiliFresh2.SP_DOSEQTY, Q_FineQty => #Dose_ChiliFresh2.SP_FINEQTY, Q_StopQty => #Dose_ChiliFresh2.r_STOP, Q_P_Speed => #Dose_ChiliFresh2.SP_IdleSPEED, Q_P_FineSpeed => #Dose_ChiliFresh2.SP_FINESPEED, Q_P_CoasSpeed => #Dose_ChiliFresh2.SP_COARSESPEED)
   END_RUNG
   // the same network as SCL:
   #SP_ChiliFresh2(CountReset := #Dose_ChiliFresh2.COUNT_RESET,   // "RawDose"
                   DoseRun := #Dose_ChiliFresh2.QDOSERun,
                   CmdStep := #Dose_ChiliFresh2.CMD_STEP,
                   FT_Tot := "Totalizer_FT-07.01".total,
                   Q_FT_Tot => #Dose_ChiliFresh2.ACT_QTY,
                   Q_SPQty => #Dose_ChiliFresh2.SP_DOSEQTY,
                   Q_FineQty => #Dose_ChiliFresh2.SP_FINEQTY,
                   Q_StopQty => #Dose_ChiliFresh2.r_STOP,
                   Q_P_Speed => #Dose_ChiliFresh2.SP_IdleSPEED,
                   Q_P_FineSpeed => #Dose_ChiliFresh2.SP_FINESPEED,
                   Q_P_CoasSpeed => #Dose_ChiliFresh2.SP_COARSESPEED);
END_REGION

REGION Network 67: Command Dose ChiliFresh2
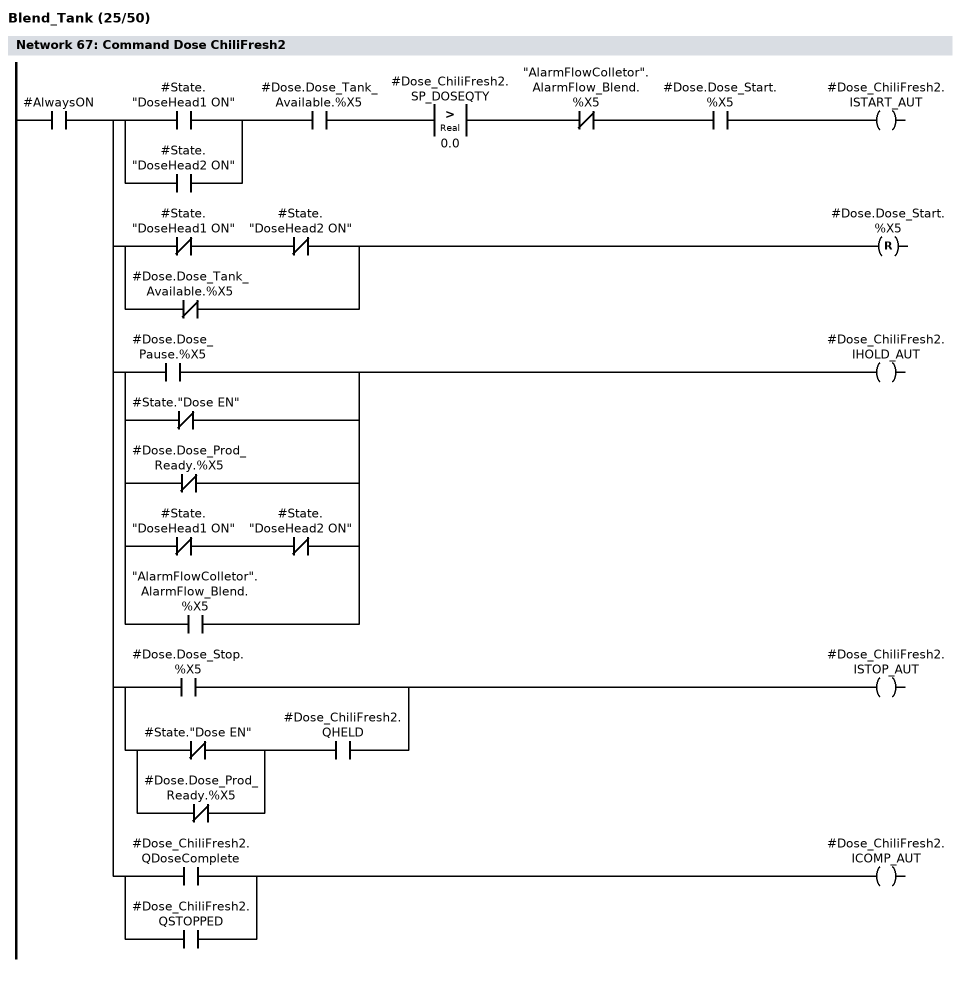
   RUNG wire#powerrail
      Contact( #AlwaysON )
      wire#w1
      Contact( #State."DoseHead1 ON" )
      wire#w2
      Contact( #Dose.Dose_Tank_Available.%X5 )
      { S7_Templates := "SrcType := Real" } GT_Contact(in1 := #Dose_ChiliFresh2.SP_DOSEQTY, in2 := 0.0)
      I_Contact( "AlarmFlowColletor".AlarmFlow_Blend.%X5 )
      Contact( #Dose.Dose_Start.%X5 )
      Coil( #Dose_ChiliFresh2.ISTART_AUT )
   END_RUNG
   RUNG wire#w1
      Contact( #State."DoseHead2 ON" )
   END_RUNG wire#w2
   RUNG wire#w1
      I_Contact( #State."DoseHead1 ON" )
      I_Contact( #State."DoseHead2 ON" )
      wire#w3
      R_Coil( #Dose.Dose_Start.%X5 )
   END_RUNG
   RUNG wire#w1
      I_Contact( #Dose.Dose_Tank_Available.%X5 )
   END_RUNG wire#w3
   RUNG wire#w1
      Contact( #Dose.Dose_Pause.%X5 )
      wire#w4
      Coil( #Dose_ChiliFresh2.IHOLD_AUT )
   END_RUNG
   RUNG wire#w1
      I_Contact( #State."Dose EN" )
   END_RUNG wire#w4
   RUNG wire#w1
      I_Contact( #Dose.Dose_Prod_Ready.%X5 )
   END_RUNG wire#w4
   RUNG wire#w1
      I_Contact( #State."DoseHead1 ON" )
      I_Contact( #State."DoseHead2 ON" )
   END_RUNG wire#w4
   RUNG wire#w1
      Contact( "AlarmFlowColletor".AlarmFlow_Blend.%X5 )
   END_RUNG wire#w4
   RUNG wire#w1
      Contact( #Dose.Dose_Stop.%X5 )
      wire#w5
      Coil( #Dose_ChiliFresh2.ISTOP_AUT )
   END_RUNG
   RUNG wire#w1
      I_Contact( #State."Dose EN" )
      wire#w6
      Contact( #Dose_ChiliFresh2.QHELD )
   END_RUNG wire#w5
   RUNG wire#w1
      I_Contact( #Dose.Dose_Prod_Ready.%X5 )
   END_RUNG wire#w6
   RUNG wire#w1
      Contact( #Dose_ChiliFresh2.QDoseComplete )
      wire#w7
      Coil( #Dose_ChiliFresh2.ICOMP_AUT )
   END_RUNG
   RUNG wire#w1
      Contact( #Dose_ChiliFresh2.QSTOPPED )
   END_RUNG wire#w7
   // the same network as SCL:
   #Dose_ChiliFresh2.ISTART_AUT := #AlwaysON AND (#State."DoseHead1 ON" OR #State."DoseHead2 ON") AND #Dose.Dose_Tank_Available.%X5 AND (#Dose_ChiliFresh2.SP_DOSEQTY > 0.0) AND NOT "AlarmFlowColletor".AlarmFlow_Blend.%X5 AND #Dose.Dose_Start.%X5;
   IF #AlwaysON AND ((NOT #State."DoseHead1 ON" AND NOT #State."DoseHead2 ON") OR NOT #Dose.Dose_Tank_Available.%X5) THEN
       #Dose.Dose_Start.%X5 := FALSE;
   END_IF;
   #Dose_ChiliFresh2.IHOLD_AUT := #AlwaysON AND (#Dose.Dose_Pause.%X5 OR NOT #State."Dose EN" OR NOT #Dose.Dose_Prod_Ready.%X5 OR (NOT #State."DoseHead1 ON" AND NOT #State."DoseHead2 ON") OR "AlarmFlowColletor".AlarmFlow_Blend.%X5);
   #Dose_ChiliFresh2.ISTOP_AUT := #AlwaysON AND (#Dose.Dose_Stop.%X5 OR ((NOT #State."Dose EN" OR NOT #Dose.Dose_Prod_Ready.%X5) AND #Dose_ChiliFresh2.QHELD));
   #Dose_ChiliFresh2.ICOMP_AUT := #AlwaysON AND (#Dose_ChiliFresh2.QDoseComplete OR #Dose_ChiliFresh2.QSTOPPED);
END_REGION

REGION Network 68: Dose ChiliFresh2
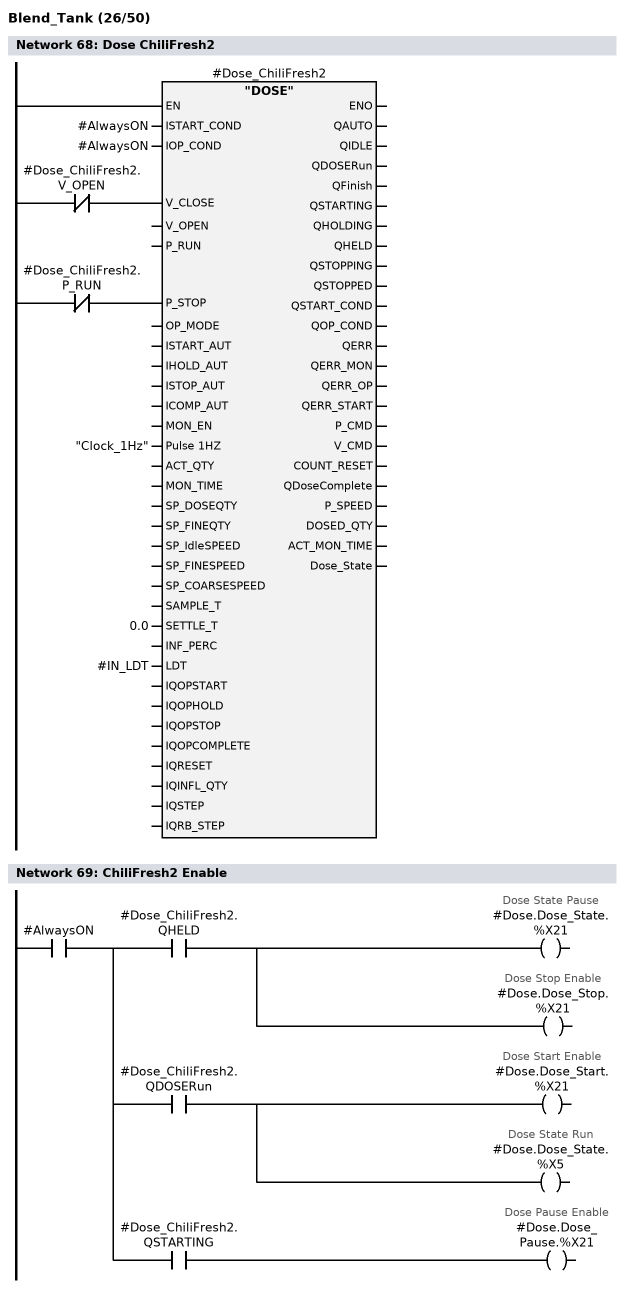
   RUNG wire#powerrail
      #Dose_ChiliFresh2(V_CLOSE := wire#w1, P_STOP := wire#w2, ISTART_COND := #AlwaysON, IOP_COND := #AlwaysON, V_OPEN :=, P_RUN :=, OP_MODE :=, ISTART_AUT :=, IHOLD_AUT :=, ISTOP_AUT :=, ICOMP_AUT :=, MON_EN :=, "Pulse 1HZ" := "Clock_1Hz", ACT_QTY :=, MON_TIME :=, SP_DOSEQTY :=, SP_FINEQTY :=, SP_IdleSPEED :=, SP_FINESPEED :=, SP_COARSESPEED :=, SAMPLE_T :=, SETTLE_T := 0.0, INF_PERC :=, LDT := #IN_LDT, IQOPSTART :=, IQOPHOLD :=, IQOPSTOP :=, IQOPCOMPLETE :=, IQRESET :=, IQINFL_QTY :=, IQSTEP :=, IQRB_STEP :=, QAUTO =>, QIDLE =>, QDOSERun =>, QFinish =>, QSTARTING =>, QHOLDING =>, QHELD =>, QSTOPPING =>, QSTOPPED =>, QSTART_COND =>, QOP_COND =>, QERR =>, QERR_MON =>, QERR_OP =>, QERR_START =>, P_CMD =>, V_CMD =>, COUNT_RESET =>, QDoseComplete =>, P_SPEED =>, DOSED_QTY =>, ACT_MON_TIME =>, Dose_State =>)
   END_RUNG
   RUNG wire#powerrail
      I_Contact( #Dose_ChiliFresh2.V_OPEN )
   END_RUNG wire#w1
   RUNG wire#powerrail
      I_Contact( #Dose_ChiliFresh2.P_RUN )
   END_RUNG wire#w2
   // the same network as SCL:
   #Dose_ChiliFresh2(ISTART_COND := #AlwaysON,   // "DOSE"
                     IOP_COND := #AlwaysON,
                     V_CLOSE := NOT #Dose_ChiliFresh2.V_OPEN,
                     P_STOP := NOT #Dose_ChiliFresh2.P_RUN,
                     "Pulse 1HZ" := "Clock_1Hz",
                     SETTLE_T := 0.0,
                     LDT := #IN_LDT);
END_REGION

REGION Network 69: ChiliFresh2 Enable
   RUNG wire#powerrail
      Contact( #AlwaysON )
      wire#w1
      Contact( #Dose_ChiliFresh2.QHELD )
      wire#w2
      Coil( #Dose.Dose_State.%X21 )   // Dose State Pause
   END_RUNG
   RUNG wire#w2
      Coil( #Dose.Dose_Stop.%X21 )   // Dose Stop Enable
   END_RUNG
   RUNG wire#w1
      Contact( #Dose_ChiliFresh2.QDOSERun )
      wire#w3
      Coil( #Dose.Dose_Start.%X21 )   // Dose Start Enable
   END_RUNG
   RUNG wire#w3
      Coil( #Dose.Dose_State.%X5 )   // Dose State Run
   END_RUNG
   RUNG wire#w1
      Contact( #Dose_ChiliFresh2.QSTARTING )
      Coil( #Dose.Dose_Pause.%X21 )   // Dose Pause Enable
   END_RUNG
   // the same network as SCL:
   #Dose.Dose_State.%X21 := #AlwaysON AND #Dose_ChiliFresh2.QHELD;   // Dose State Pause
   #Dose.Dose_Stop.%X21 := #Dose.Dose_State.%X21;   // Dose Stop Enable
   #Dose.Dose_Start.%X21 := #AlwaysON AND #Dose_ChiliFresh2.QDOSERun;   // Dose Start Enable
   #Dose.Dose_State.%X5 := #Dose.Dose_Start.%X21;   // Dose State Run
   #Dose.Dose_Pause.%X21 := #AlwaysON AND #Dose_ChiliFresh2.QSTARTING;   // Dose Pause Enable
END_REGION

REGION Network 70: ChiliFresh2 Header Req
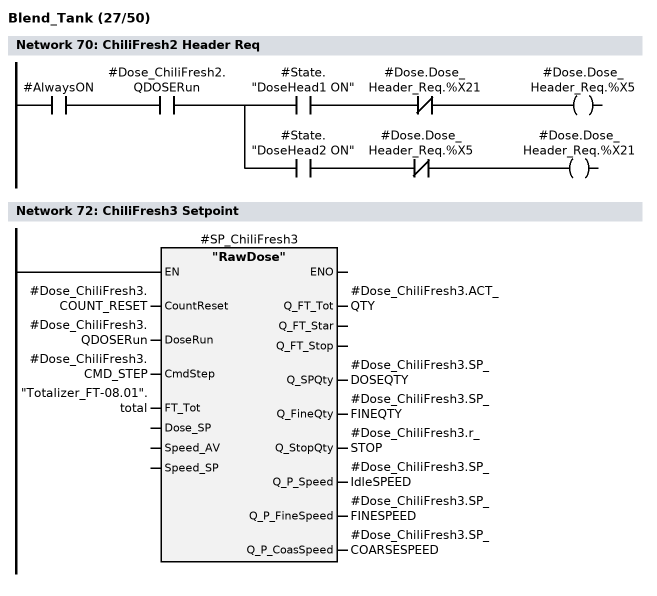
   RUNG wire#powerrail
      Contact( #AlwaysON )
      Contact( #Dose_ChiliFresh2.QDOSERun )
      wire#w1
      Contact( #State."DoseHead1 ON" )
      I_Contact( #Dose.Dose_Header_Req.%X21 )
      Coil( #Dose.Dose_Header_Req.%X5 )
   END_RUNG
   RUNG wire#w1
      Contact( #State."DoseHead2 ON" )
      I_Contact( #Dose.Dose_Header_Req.%X5 )
      Coil( #Dose.Dose_Header_Req.%X21 )
   END_RUNG
   // the same network as SCL:
   #_w1 := #AlwaysON AND #Dose_ChiliFresh2.QDOSERun;
   #Dose.Dose_Header_Req.%X5 := #_w1 AND #State."DoseHead1 ON" AND NOT #Dose.Dose_Header_Req.%X21;
   #Dose.Dose_Header_Req.%X21 := #_w1 AND #State."DoseHead2 ON" AND NOT #Dose.Dose_Header_Req.%X5;
END_REGION

REGION Network 72: ChiliFresh3 Setpoint
   RUNG wire#powerrail
      #SP_ChiliFresh3(CountReset := #Dose_ChiliFresh3.COUNT_RESET, DoseRun := #Dose_ChiliFresh3.QDOSERun, CmdStep := #Dose_ChiliFresh3.CMD_STEP, FT_Tot := "Totalizer_FT-08.01".total, Dose_SP :=, Speed_AV :=, Speed_SP :=, Q_FT_Tot => #Dose_ChiliFresh3.ACT_QTY, Q_FT_Star =>, Q_FT_Stop =>, Q_SPQty => #Dose_ChiliFresh3.SP_DOSEQTY, Q_FineQty => #Dose_ChiliFresh3.SP_FINEQTY, Q_StopQty => #Dose_ChiliFresh3.r_STOP, Q_P_Speed => #Dose_ChiliFresh3.SP_IdleSPEED, Q_P_FineSpeed => #Dose_ChiliFresh3.SP_FINESPEED, Q_P_CoasSpeed => #Dose_ChiliFresh3.SP_COARSESPEED)
   END_RUNG
   // the same network as SCL:
   #SP_ChiliFresh3(CountReset := #Dose_ChiliFresh3.COUNT_RESET,   // "RawDose"
                   DoseRun := #Dose_ChiliFresh3.QDOSERun,
                   CmdStep := #Dose_ChiliFresh3.CMD_STEP,
                   FT_Tot := "Totalizer_FT-08.01".total,
                   Q_FT_Tot => #Dose_ChiliFresh3.ACT_QTY,
                   Q_SPQty => #Dose_ChiliFresh3.SP_DOSEQTY,
                   Q_FineQty => #Dose_ChiliFresh3.SP_FINEQTY,
                   Q_StopQty => #Dose_ChiliFresh3.r_STOP,
                   Q_P_Speed => #Dose_ChiliFresh3.SP_IdleSPEED,
                   Q_P_FineSpeed => #Dose_ChiliFresh3.SP_FINESPEED,
                   Q_P_CoasSpeed => #Dose_ChiliFresh3.SP_COARSESPEED);
END_REGION

REGION Network 73: Command Dose ChiliFresh3
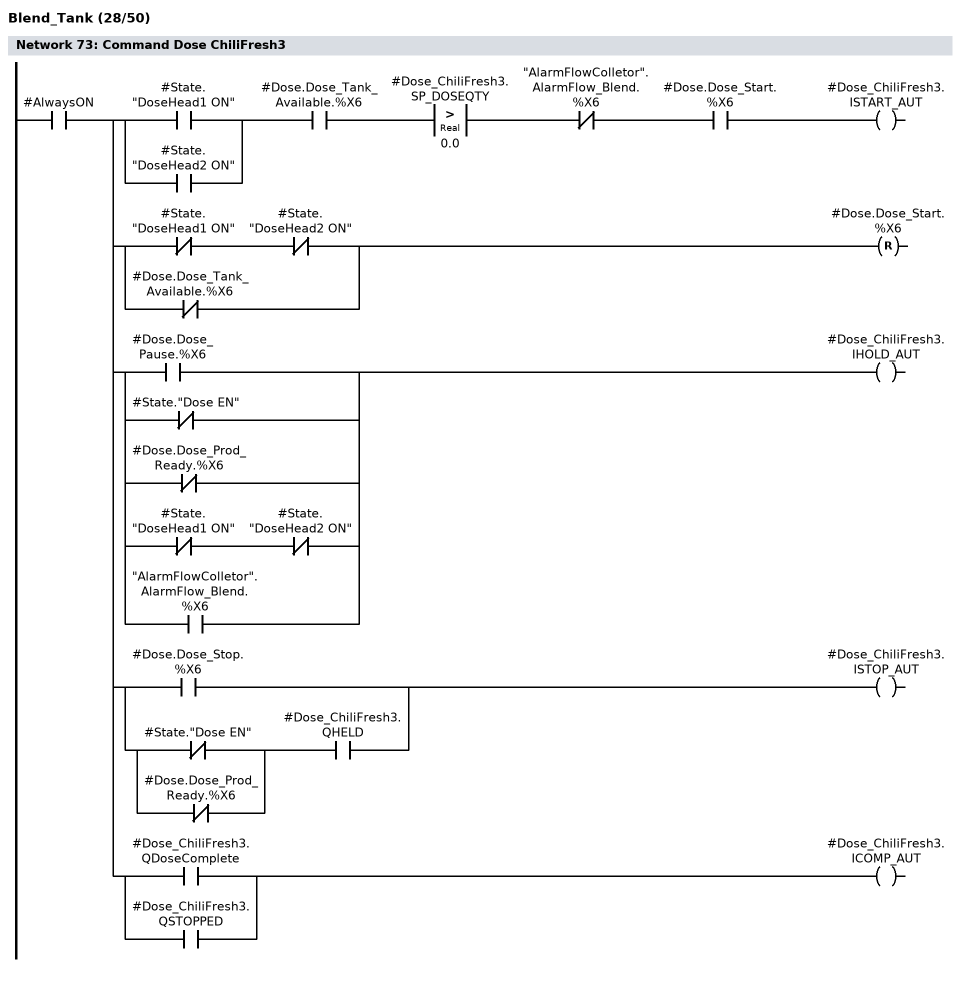
   RUNG wire#powerrail
      Contact( #AlwaysON )
      wire#w1
      Contact( #State."DoseHead1 ON" )
      wire#w2
      Contact( #Dose.Dose_Tank_Available.%X6 )
      { S7_Templates := "SrcType := Real" } GT_Contact(in1 := #Dose_ChiliFresh3.SP_DOSEQTY, in2 := 0.0)
      I_Contact( "AlarmFlowColletor".AlarmFlow_Blend.%X6 )
      Contact( #Dose.Dose_Start.%X6 )
      Coil( #Dose_ChiliFresh3.ISTART_AUT )
   END_RUNG
   RUNG wire#w1
      Contact( #State."DoseHead2 ON" )
   END_RUNG wire#w2
   RUNG wire#w1
      I_Contact( #State."DoseHead1 ON" )
      I_Contact( #State."DoseHead2 ON" )
      wire#w3
      R_Coil( #Dose.Dose_Start.%X6 )
   END_RUNG
   RUNG wire#w1
      I_Contact( #Dose.Dose_Tank_Available.%X6 )
   END_RUNG wire#w3
   RUNG wire#w1
      Contact( #Dose.Dose_Pause.%X6 )
      wire#w4
      Coil( #Dose_ChiliFresh3.IHOLD_AUT )
   END_RUNG
   RUNG wire#w1
      I_Contact( #State."Dose EN" )
   END_RUNG wire#w4
   RUNG wire#w1
      I_Contact( #Dose.Dose_Prod_Ready.%X6 )
   END_RUNG wire#w4
   RUNG wire#w1
      I_Contact( #State."DoseHead1 ON" )
      I_Contact( #State."DoseHead2 ON" )
   END_RUNG wire#w4
   RUNG wire#w1
      Contact( "AlarmFlowColletor".AlarmFlow_Blend.%X6 )
   END_RUNG wire#w4
   RUNG wire#w1
      Contact( #Dose.Dose_Stop.%X6 )
      wire#w5
      Coil( #Dose_ChiliFresh3.ISTOP_AUT )
   END_RUNG
   RUNG wire#w1
      I_Contact( #State."Dose EN" )
      wire#w6
      Contact( #Dose_ChiliFresh3.QHELD )
   END_RUNG wire#w5
   RUNG wire#w1
      I_Contact( #Dose.Dose_Prod_Ready.%X6 )
   END_RUNG wire#w6
   RUNG wire#w1
      Contact( #Dose_ChiliFresh3.QDoseComplete )
      wire#w7
      Coil( #Dose_ChiliFresh3.ICOMP_AUT )
   END_RUNG
   RUNG wire#w1
      Contact( #Dose_ChiliFresh3.QSTOPPED )
   END_RUNG wire#w7
   // the same network as SCL:
   #Dose_ChiliFresh3.ISTART_AUT := #AlwaysON AND (#State."DoseHead1 ON" OR #State."DoseHead2 ON") AND #Dose.Dose_Tank_Available.%X6 AND (#Dose_ChiliFresh3.SP_DOSEQTY > 0.0) AND NOT "AlarmFlowColletor".AlarmFlow_Blend.%X6 AND #Dose.Dose_Start.%X6;
   IF #AlwaysON AND ((NOT #State."DoseHead1 ON" AND NOT #State."DoseHead2 ON") OR NOT #Dose.Dose_Tank_Available.%X6) THEN
       #Dose.Dose_Start.%X6 := FALSE;
   END_IF;
   #Dose_ChiliFresh3.IHOLD_AUT := #AlwaysON AND (#Dose.Dose_Pause.%X6 OR NOT #State."Dose EN" OR NOT #Dose.Dose_Prod_Ready.%X6 OR (NOT #State."DoseHead1 ON" AND NOT #State."DoseHead2 ON") OR "AlarmFlowColletor".AlarmFlow_Blend.%X6);
   #Dose_ChiliFresh3.ISTOP_AUT := #AlwaysON AND (#Dose.Dose_Stop.%X6 OR ((NOT #State."Dose EN" OR NOT #Dose.Dose_Prod_Ready.%X6) AND #Dose_ChiliFresh3.QHELD));
   #Dose_ChiliFresh3.ICOMP_AUT := #AlwaysON AND (#Dose_ChiliFresh3.QDoseComplete OR #Dose_ChiliFresh3.QSTOPPED);
END_REGION

REGION Network 74: Dose ChiliFresh3
